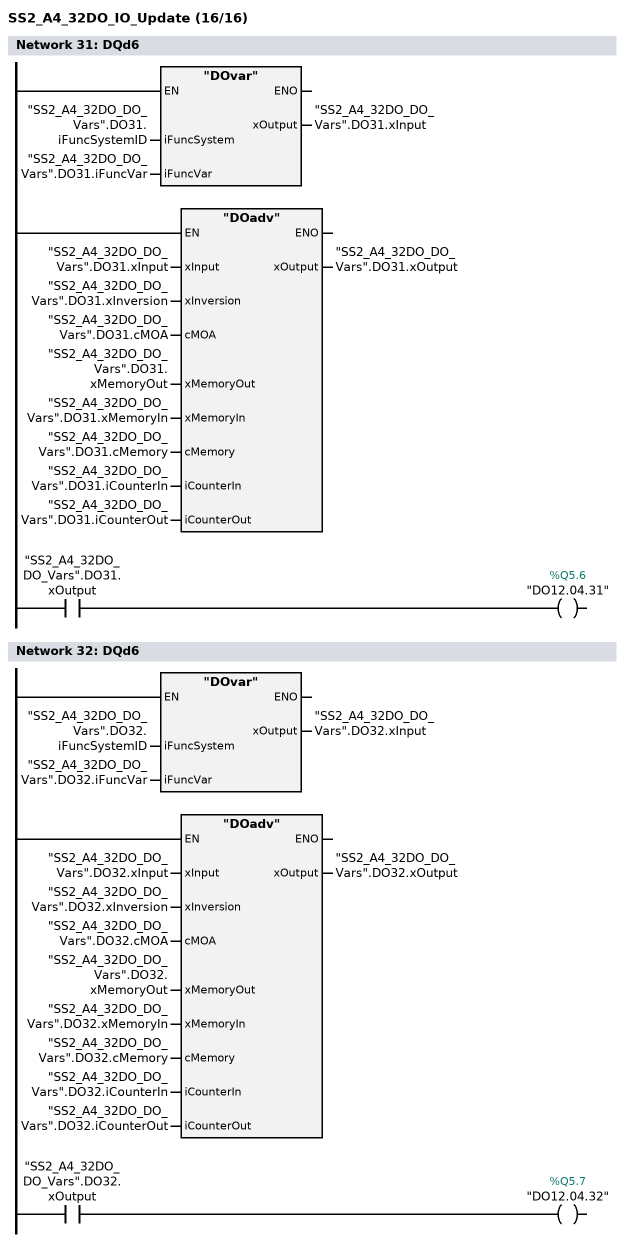
   RUNG wire#powerrail
      "DOvar"(iFuncSystem := "SS2_A4_32DO_DO_Vars".DO31.iFuncSystemID, iFuncVar := "SS2_A4_32DO_DO_Vars".DO31.iFuncVar, xOutput => "SS2_A4_32DO_DO_Vars".DO31.xInput)
   END_RUNG
   RUNG wire#powerrail
      "DOadv"(xInput := "SS2_A4_32DO_DO_Vars".DO31.xInput, xInversion := "SS2_A4_32DO_DO_Vars".DO31.xInversion, cMOA := "SS2_A4_32DO_DO_Vars".DO31.cMOA, xMemoryOut := "SS2_A4_32DO_DO_Vars".DO31.xMemoryOut, xMemoryIn := "SS2_A4_32DO_DO_Vars".DO31.xMemoryIn, cMemory := "SS2_A4_32DO_DO_Vars".DO31.cMemory, iCounterIn := "SS2_A4_32DO_DO_Vars".DO31.iCounterIn, iCounterOut := "SS2_A4_32DO_DO_Vars".DO31.iCounterOut, xOutput => "SS2_A4_32DO_DO_Vars".DO31.xOutput)
   END_RUNG
   RUNG wire#powerrail
      Contact( "SS2_A4_32DO_DO_Vars".DO31.xOutput )
      Coil( "DO12.04.31" )
   END_RUNG
   // the same network as SCL:
   "DOvar"(iFuncSystem := "SS2_A4_32DO_DO_Vars".DO31.iFuncSystemID,
           iFuncVar := "SS2_A4_32DO_DO_Vars".DO31.iFuncVar,
           xOutput => "SS2_A4_32DO_DO_Vars".DO31.xInput);
   "DOadv"(xInput := "SS2_A4_32DO_DO_Vars".DO31.xInput,
           xInversion := "SS2_A4_32DO_DO_Vars".DO31.xInversion,
           cMOA := "SS2_A4_32DO_DO_Vars".DO31.cMOA,
           xMemoryOut := "SS2_A4_32DO_DO_Vars".DO31.xMemoryOut,
           xMemoryIn := "SS2_A4_32DO_DO_Vars".DO31.xMemoryIn,
           cMemory := "SS2_A4_32DO_DO_Vars".DO31.cMemory,
           iCounterIn := "SS2_A4_32DO_DO_Vars".DO31.iCounterIn,
           iCounterOut := "SS2_A4_32DO_DO_Vars".DO31.iCounterOut,
           xOutput => "SS2_A4_32DO_DO_Vars".DO31.xOutput);
   "DO12.04.31" := "SS2_A4_32DO_DO_Vars".DO31.xOutput;
END_REGION

REGION Network 32: DQd6
   RUNG wire#powerrail
      "DOvar"(iFuncSystem := "SS2_A4_32DO_DO_Vars".DO32.iFuncSystemID, iFuncVar := "SS2_A4_32DO_DO_Vars".DO32.iFuncVar, xOutput => "SS2_A4_32DO_DO_Vars".DO32.xInput)
   END_RUNG
   RUNG wire#powerrail
      "DOadv"(xInput := "SS2_A4_32DO_DO_Vars".DO32.xInput, xInversion := "SS2_A4_32DO_DO_Vars".DO32.xInversion, cMOA := "SS2_A4_32DO_DO_Vars".DO32.cMOA, xMemoryOut := "SS2_A4_32DO_DO_Vars".DO32.xMemoryOut, xMemoryIn := "SS2_A4_32DO_DO_Vars".DO32.xMemoryIn, cMemory := "SS2_A4_32DO_DO_Vars".DO32.cMemory, iCounterIn := "SS2_A4_32DO_DO_Vars".DO32.iCounterIn, iCounterOut := "SS2_A4_32DO_DO_Vars".DO32.iCounterOut, xOutput => "SS2_A4_32DO_DO_Vars".DO32.xOutput)
   END_RUNG
   RUNG wire#powerrail
      Contact( "SS2_A4_32DO_DO_Vars".DO32.xOutput )
      Coil( "DO12.04.32" )
   END_RUNG
   // the same network as SCL:
   "DOvar"(iFuncSystem := "SS2_A4_32DO_DO_Vars".DO32.iFuncSystemID,
           iFuncVar := "SS2_A4_32DO_DO_Vars".DO32.iFuncVar,
           xOutput => "SS2_A4_32DO_DO_Vars".DO32.xInput);
   "DOadv"(xInput := "SS2_A4_32DO_DO_Vars".DO32.xInput,
           xInversion := "SS2_A4_32DO_DO_Vars".DO32.xInversion,
           cMOA := "SS2_A4_32DO_DO_Vars".DO32.cMOA,
           xMemoryOut := "SS2_A4_32DO_DO_Vars".DO32.xMemoryOut,
           xMemoryIn := "SS2_A4_32DO_DO_Vars".DO32.xMemoryIn,
           cMemory := "SS2_A4_32DO_DO_Vars".DO32.cMemory,
           iCounterIn := "SS2_A4_32DO_DO_Vars".DO32.iCounterIn,
           iCounterOut := "SS2_A4_32DO_DO_Vars".DO32.iCounterOut,
           xOutput => "SS2_A4_32DO_DO_Vars".DO32.xOutput);
   "DO12.04.32" := "SS2_A4_32DO_DO_Vars".DO32.xOutput;
END_REGION
END_FUNCTION

FUNCTION "SS2_A5_16DI_IO_Update" : Void   // FC11160, LAD
{ S7_Optimized_Access := 'TRUE' }
VERSION : 0.1
// stored: AutoNumber false, IsIECCheckEnabled false, SetENOAutomatically false, UDAEnableTagReadback false
BEGIN

REGION Network 1: DIa0
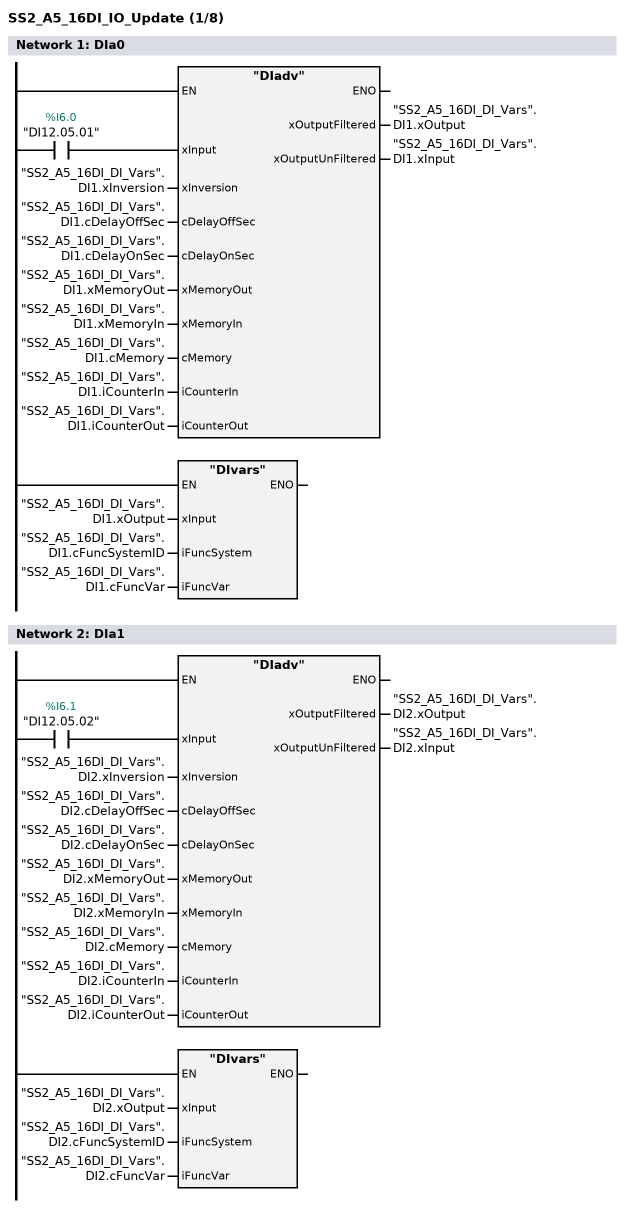
   RUNG wire#powerrail
      "DIadv"(xInput := wire#w1, xInversion := "SS2_A5_16DI_DI_Vars".DI1.xInversion, cDelayOffSec := "SS2_A5_16DI_DI_Vars".DI1.cDelayOffSec, cDelayOnSec := "SS2_A5_16DI_DI_Vars".DI1.cDelayOnSec, xMemoryOut := "SS2_A5_16DI_DI_Vars".DI1.xMemoryOut, xMemoryIn := "SS2_A5_16DI_DI_Vars".DI1.xMemoryIn, cMemory := "SS2_A5_16DI_DI_Vars".DI1.cMemory, xOutputFiltered => "SS2_A5_16DI_DI_Vars".DI1.xOutput, xOutputUnFiltered => "SS2_A5_16DI_DI_Vars".DI1.xInput, iCounterIn := "SS2_A5_16DI_DI_Vars".DI1.iCounterIn, iCounterOut := "SS2_A5_16DI_DI_Vars".DI1.iCounterOut)
   END_RUNG
   RUNG wire#powerrail
      Contact( "DI12.05.01" )
   END_RUNG wire#w1
   RUNG wire#powerrail
      "DIvars"(xInput := "SS2_A5_16DI_DI_Vars".DI1.xOutput, iFuncSystem := "SS2_A5_16DI_DI_Vars".DI1.cFuncSystemID, iFuncVar := "SS2_A5_16DI_DI_Vars".DI1.cFuncVar)
   END_RUNG
   // the same network as SCL:
   "DIadv"(xInput := "DI12.05.01",
           xInversion := "SS2_A5_16DI_DI_Vars".DI1.xInversion,
           cDelayOffSec := "SS2_A5_16DI_DI_Vars".DI1.cDelayOffSec,
           cDelayOnSec := "SS2_A5_16DI_DI_Vars".DI1.cDelayOnSec,
           xMemoryOut := "SS2_A5_16DI_DI_Vars".DI1.xMemoryOut,
           xMemoryIn := "SS2_A5_16DI_DI_Vars".DI1.xMemoryIn,
           cMemory := "SS2_A5_16DI_DI_Vars".DI1.cMemory,
           iCounterIn := "SS2_A5_16DI_DI_Vars".DI1.iCounterIn,
           iCounterOut := "SS2_A5_16DI_DI_Vars".DI1.iCounterOut,
           xOutputFiltered => "SS2_A5_16DI_DI_Vars".DI1.xOutput,
           xOutputUnFiltered => "SS2_A5_16DI_DI_Vars".DI1.xInput);
   "DIvars"(xInput := "SS2_A5_16DI_DI_Vars".DI1.xOutput,
            iFuncSystem := "SS2_A5_16DI_DI_Vars".DI1.cFuncSystemID,
            iFuncVar := "SS2_A5_16DI_DI_Vars".DI1.cFuncVar);
END_REGION

REGION Network 2: DIa1
   RUNG wire#powerrail
      "DIadv"(xInput := wire#w1, xInversion := "SS2_A5_16DI_DI_Vars".DI2.xInversion, cDelayOffSec := "SS2_A5_16DI_DI_Vars".DI2.cDelayOffSec, cDelayOnSec := "SS2_A5_16DI_DI_Vars".DI2.cDelayOnSec, xMemoryOut := "SS2_A5_16DI_DI_Vars".DI2.xMemoryOut, xMemoryIn := "SS2_A5_16DI_DI_Vars".DI2.xMemoryIn, cMemory := "SS2_A5_16DI_DI_Vars".DI2.cMemory, xOutputFiltered => "SS2_A5_16DI_DI_Vars".DI2.xOutput, xOutputUnFiltered => "SS2_A5_16DI_DI_Vars".DI2.xInput, iCounterIn := "SS2_A5_16DI_DI_Vars".DI2.iCounterIn, iCounterOut := "SS2_A5_16DI_DI_Vars".DI2.iCounterOut)
   END_RUNG
   RUNG wire#powerrail
      Contact( "DI12.05.02" )
   END_RUNG wire#w1
   RUNG wire#powerrail
      "DIvars"(xInput := "SS2_A5_16DI_DI_Vars".DI2.xOutput, iFuncSystem := "SS2_A5_16DI_DI_Vars".DI2.cFuncSystemID, iFuncVar := "SS2_A5_16DI_DI_Vars".DI2.cFuncVar)
   END_RUNG
   // the same network as SCL:
   "DIadv"(xInput := "DI12.05.02",
           xInversion := "SS2_A5_16DI_DI_Vars".DI2.xInversion,
           cDelayOffSec := "SS2_A5_16DI_DI_Vars".DI2.cDelayOffSec,
           cDelayOnSec := "SS2_A5_16DI_DI_Vars".DI2.cDelayOnSec,
           xMemoryOut := "SS2_A5_16DI_DI_Vars".DI2.xMemoryOut,
           xMemoryIn := "SS2_A5_16DI_DI_Vars".DI2.xMemoryIn,
           cMemory := "SS2_A5_16DI_DI_Vars".DI2.cMemory,
           iCounterIn := "SS2_A5_16DI_DI_Vars".DI2.iCounterIn,
           iCounterOut := "SS2_A5_16DI_DI_Vars".DI2.iCounterOut,
           xOutputFiltered => "SS2_A5_16DI_DI_Vars".DI2.xOutput,
           xOutputUnFiltered => "SS2_A5_16DI_DI_Vars".DI2.xInput);
   "DIvars"(xInput := "SS2_A5_16DI_DI_Vars".DI2.xOutput,
            iFuncSystem := "SS2_A5_16DI_DI_Vars".DI2.cFuncSystemID,
            iFuncVar := "SS2_A5_16DI_DI_Vars".DI2.cFuncVar);
END_REGION

REGION Network 3: DIa2
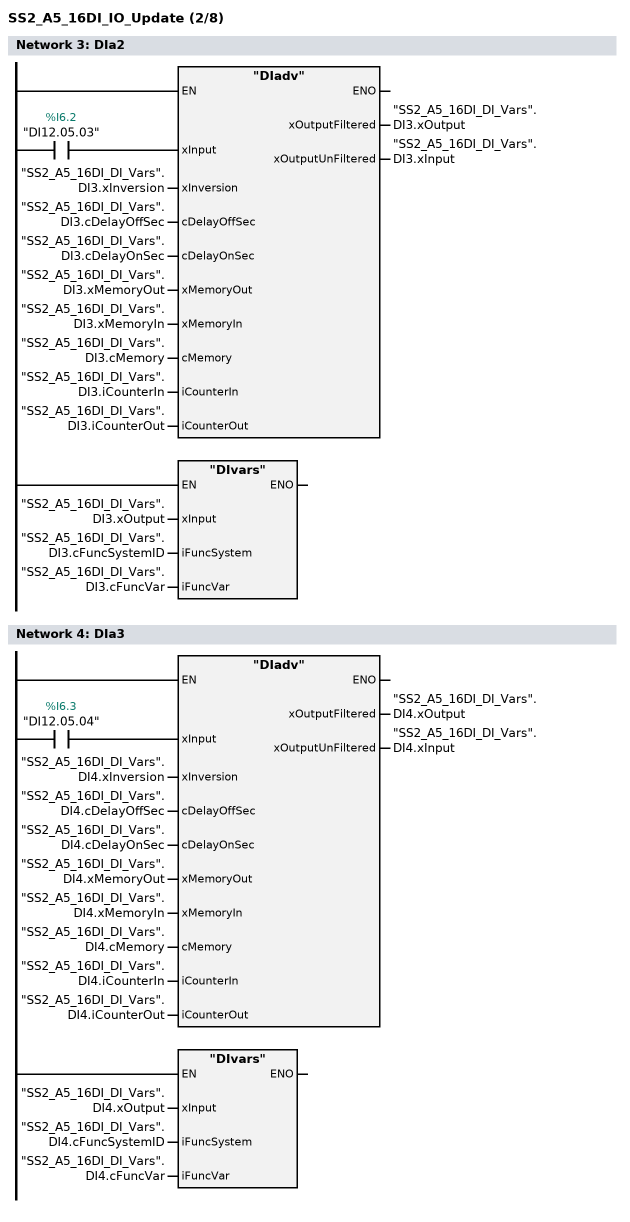
   RUNG wire#powerrail
      "DIadv"(xInput := wire#w1, xInversion := "SS2_A5_16DI_DI_Vars".DI3.xInversion, cDelayOffSec := "SS2_A5_16DI_DI_Vars".DI3.cDelayOffSec, cDelayOnSec := "SS2_A5_16DI_DI_Vars".DI3.cDelayOnSec, xMemoryOut := "SS2_A5_16DI_DI_Vars".DI3.xMemoryOut, xMemoryIn := "SS2_A5_16DI_DI_Vars".DI3.xMemoryIn, cMemory := "SS2_A5_16DI_DI_Vars".DI3.cMemory, xOutputFiltered => "SS2_A5_16DI_DI_Vars".DI3.xOutput, xOutputUnFiltered => "SS2_A5_16DI_DI_Vars".DI3.xInput, iCounterIn := "SS2_A5_16DI_DI_Vars".DI3.iCounterIn, iCounterOut := "SS2_A5_16DI_DI_Vars".DI3.iCounterOut)
   END_RUNG
   RUNG wire#powerrail
      Contact( "DI12.05.03" )
   END_RUNG wire#w1
   RUNG wire#powerrail
      "DIvars"(xInput := "SS2_A5_16DI_DI_Vars".DI3.xOutput, iFuncSystem := "SS2_A5_16DI_DI_Vars".DI3.cFuncSystemID, iFuncVar := "SS2_A5_16DI_DI_Vars".DI3.cFuncVar)
   END_RUNG
   // the same network as SCL:
   "DIadv"(xInput := "DI12.05.03",
           xInversion := "SS2_A5_16DI_DI_Vars".DI3.xInversion,
           cDelayOffSec := "SS2_A5_16DI_DI_Vars".DI3.cDelayOffSec,
           cDelayOnSec := "SS2_A5_16DI_DI_Vars".DI3.cDelayOnSec,
           xMemoryOut := "SS2_A5_16DI_DI_Vars".DI3.xMemoryOut,
           xMemoryIn := "SS2_A5_16DI_DI_Vars".DI3.xMemoryIn,
           cMemory := "SS2_A5_16DI_DI_Vars".DI3.cMemory,
           iCounterIn := "SS2_A5_16DI_DI_Vars".DI3.iCounterIn,
           iCounterOut := "SS2_A5_16DI_DI_Vars".DI3.iCounterOut,
           xOutputFiltered => "SS2_A5_16DI_DI_Vars".DI3.xOutput,
           xOutputUnFiltered => "SS2_A5_16DI_DI_Vars".DI3.xInput);
   "DIvars"(xInput := "SS2_A5_16DI_DI_Vars".DI3.xOutput,
            iFuncSystem := "SS2_A5_16DI_DI_Vars".DI3.cFuncSystemID,
            iFuncVar := "SS2_A5_16DI_DI_Vars".DI3.cFuncVar);
END_REGION

REGION Network 4: DIa3
   RUNG wire#powerrail
      "DIadv"(xInput := wire#w1, xInversion := "SS2_A5_16DI_DI_Vars".DI4.xInversion, cDelayOffSec := "SS2_A5_16DI_DI_Vars".DI4.cDelayOffSec, cDelayOnSec := "SS2_A5_16DI_DI_Vars".DI4.cDelayOnSec, xMemoryOut := "SS2_A5_16DI_DI_Vars".DI4.xMemoryOut, xMemoryIn := "SS2_A5_16DI_DI_Vars".DI4.xMemoryIn, cMemory := "SS2_A5_16DI_DI_Vars".DI4.cMemory, xOutputFiltered => "SS2_A5_16DI_DI_Vars".DI4.xOutput, xOutputUnFiltered => "SS2_A5_16DI_DI_Vars".DI4.xInput, iCounterIn := "SS2_A5_16DI_DI_Vars".DI4.iCounterIn, iCounterOut := "SS2_A5_16DI_DI_Vars".DI4.iCounterOut)
   END_RUNG
   RUNG wire#powerrail
      Contact( "DI12.05.04" )
   END_RUNG wire#w1
   RUNG wire#powerrail
      "DIvars"(xInput := "SS2_A5_16DI_DI_Vars".DI4.xOutput, iFuncSystem := "SS2_A5_16DI_DI_Vars".DI4.cFuncSystemID, iFuncVar := "SS2_A5_16DI_DI_Vars".DI4.cFuncVar)
   END_RUNG
   // the same network as SCL:
   "DIadv"(xInput := "DI12.05.04",
           xInversion := "SS2_A5_16DI_DI_Vars".DI4.xInversion,
           cDelayOffSec := "SS2_A5_16DI_DI_Vars".DI4.cDelayOffSec,
           cDelayOnSec := "SS2_A5_16DI_DI_Vars".DI4.cDelayOnSec,
           xMemoryOut := "SS2_A5_16DI_DI_Vars".DI4.xMemoryOut,
           xMemoryIn := "SS2_A5_16DI_DI_Vars".DI4.xMemoryIn,
           cMemory := "SS2_A5_16DI_DI_Vars".DI4.cMemory,
           iCounterIn := "SS2_A5_16DI_DI_Vars".DI4.iCounterIn,
           iCounterOut := "SS2_A5_16DI_DI_Vars".DI4.iCounterOut,
           xOutputFiltered => "SS2_A5_16DI_DI_Vars".DI4.xOutput,
           xOutputUnFiltered => "SS2_A5_16DI_DI_Vars".DI4.xInput);
   "DIvars"(xInput := "SS2_A5_16DI_DI_Vars".DI4.xOutput,
            iFuncSystem := "SS2_A5_16DI_DI_Vars".DI4.cFuncSystemID,
            iFuncVar := "SS2_A5_16DI_DI_Vars".DI4.cFuncVar);
END_REGION

REGION Network 5: DIa4
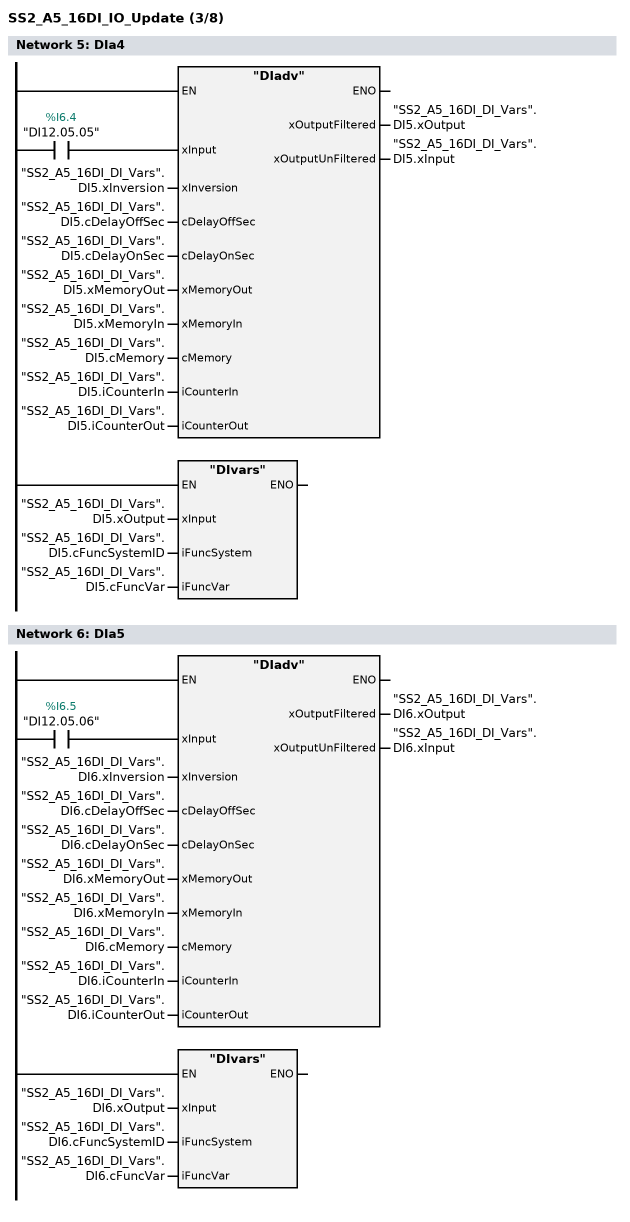
   RUNG wire#powerrail
      "DIadv"(xInput := wire#w1, xInversion := "SS2_A5_16DI_DI_Vars".DI5.xInversion, cDelayOffSec := "SS2_A5_16DI_DI_Vars".DI5.cDelayOffSec, cDelayOnSec := "SS2_A5_16DI_DI_Vars".DI5.cDelayOnSec, xMemoryOut := "SS2_A5_16DI_DI_Vars".DI5.xMemoryOut, xMemoryIn := "SS2_A5_16DI_DI_Vars".DI5.xMemoryIn, cMemory := "SS2_A5_16DI_DI_Vars".DI5.cMemory, xOutputFiltered => "SS2_A5_16DI_DI_Vars".DI5.xOutput, xOutputUnFiltered => "SS2_A5_16DI_DI_Vars".DI5.xInput, iCounterIn := "SS2_A5_16DI_DI_Vars".DI5.iCounterIn, iCounterOut := "SS2_A5_16DI_DI_Vars".DI5.iCounterOut)
   END_RUNG
   RUNG wire#powerrail
      Contact( "DI12.05.05" )
   END_RUNG wire#w1
   RUNG wire#powerrail
      "DIvars"(xInput := "SS2_A5_16DI_DI_Vars".DI5.xOutput, iFuncSystem := "SS2_A5_16DI_DI_Vars".DI5.cFuncSystemID, iFuncVar := "SS2_A5_16DI_DI_Vars".DI5.cFuncVar)
   END_RUNG
   // the same network as SCL:
   "DIadv"(xInput := "DI12.05.05",
           xInversion := "SS2_A5_16DI_DI_Vars".DI5.xInversion,
           cDelayOffSec := "SS2_A5_16DI_DI_Vars".DI5.cDelayOffSec,
           cDelayOnSec := "SS2_A5_16DI_DI_Vars".DI5.cDelayOnSec,
           xMemoryOut := "SS2_A5_16DI_DI_Vars".DI5.xMemoryOut,
           xMemoryIn := "SS2_A5_16DI_DI_Vars".DI5.xMemoryIn,
           cMemory := "SS2_A5_16DI_DI_Vars".DI5.cMemory,
           iCounterIn := "SS2_A5_16DI_DI_Vars".DI5.iCounterIn,
           iCounterOut := "SS2_A5_16DI_DI_Vars".DI5.iCounterOut,
           xOutputFiltered => "SS2_A5_16DI_DI_Vars".DI5.xOutput,
           xOutputUnFiltered => "SS2_A5_16DI_DI_Vars".DI5.xInput);
   "DIvars"(xInput := "SS2_A5_16DI_DI_Vars".DI5.xOutput,
            iFuncSystem := "SS2_A5_16DI_DI_Vars".DI5.cFuncSystemID,
            iFuncVar := "SS2_A5_16DI_DI_Vars".DI5.cFuncVar);
END_REGION

REGION Network 6: DIa5
   RUNG wire#powerrail
      "DIadv"(xInput := wire#w1, xInversion := "SS2_A5_16DI_DI_Vars".DI6.xInversion, cDelayOffSec := "SS2_A5_16DI_DI_Vars".DI6.cDelayOffSec, cDelayOnSec := "SS2_A5_16DI_DI_Vars".DI6.cDelayOnSec, xMemoryOut := "SS2_A5_16DI_DI_Vars".DI6.xMemoryOut, xMemoryIn := "SS2_A5_16DI_DI_Vars".DI6.xMemoryIn, cMemory := "SS2_A5_16DI_DI_Vars".DI6.cMemory, xOutputFiltered => "SS2_A5_16DI_DI_Vars".DI6.xOutput, xOutputUnFiltered => "SS2_A5_16DI_DI_Vars".DI6.xInput, iCounterIn := "SS2_A5_16DI_DI_Vars".DI6.iCounterIn, iCounterOut := "SS2_A5_16DI_DI_Vars".DI6.iCounterOut)
   END_RUNG
   RUNG wire#powerrail
      Contact( "DI12.05.06" )
   END_RUNG wire#w1
   RUNG wire#powerrail
      "DIvars"(xInput := "SS2_A5_16DI_DI_Vars".DI6.xOutput, iFuncSystem := "SS2_A5_16DI_DI_Vars".DI6.cFuncSystemID, iFuncVar := "SS2_A5_16DI_DI_Vars".DI6.cFuncVar)
   END_RUNG
   // the same network as SCL:
   "DIadv"(xInput := "DI12.05.06",
           xInversion := "SS2_A5_16DI_DI_Vars".DI6.xInversion,
           cDelayOffSec := "SS2_A5_16DI_DI_Vars".DI6.cDelayOffSec,
           cDelayOnSec := "SS2_A5_16DI_DI_Vars".DI6.cDelayOnSec,
           xMemoryOut := "SS2_A5_16DI_DI_Vars".DI6.xMemoryOut,
           xMemoryIn := "SS2_A5_16DI_DI_Vars".DI6.xMemoryIn,
           cMemory := "SS2_A5_16DI_DI_Vars".DI6.cMemory,
           iCounterIn := "SS2_A5_16DI_DI_Vars".DI6.iCounterIn,
           iCounterOut := "SS2_A5_16DI_DI_Vars".DI6.iCounterOut,
           xOutputFiltered => "SS2_A5_16DI_DI_Vars".DI6.xOutput,
           xOutputUnFiltered => "SS2_A5_16DI_DI_Vars".DI6.xInput);
   "DIvars"(xInput := "SS2_A5_16DI_DI_Vars".DI6.xOutput,
            iFuncSystem := "SS2_A5_16DI_DI_Vars".DI6.cFuncSystemID,
            iFuncVar := "SS2_A5_16DI_DI_Vars".DI6.cFuncVar);
END_REGION

REGION Network 7: DIa6
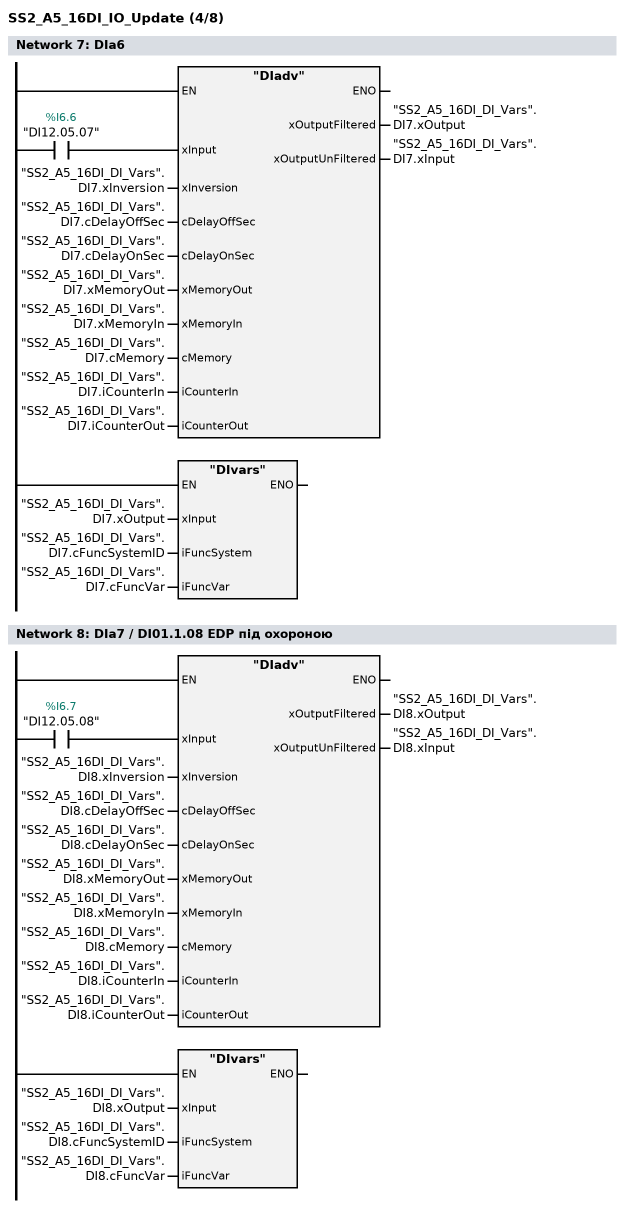
   RUNG wire#powerrail
      "DIadv"(xInput := wire#w1, xInversion := "SS2_A5_16DI_DI_Vars".DI7.xInversion, cDelayOffSec := "SS2_A5_16DI_DI_Vars".DI7.cDelayOffSec, cDelayOnSec := "SS2_A5_16DI_DI_Vars".DI7.cDelayOnSec, xMemoryOut := "SS2_A5_16DI_DI_Vars".DI7.xMemoryOut, xMemoryIn := "SS2_A5_16DI_DI_Vars".DI7.xMemoryIn, cMemory := "SS2_A5_16DI_DI_Vars".DI7.cMemory, xOutputFiltered => "SS2_A5_16DI_DI_Vars".DI7.xOutput, xOutputUnFiltered => "SS2_A5_16DI_DI_Vars".DI7.xInput, iCounterIn := "SS2_A5_16DI_DI_Vars".DI7.iCounterIn, iCounterOut := "SS2_A5_16DI_DI_Vars".DI7.iCounterOut)
   END_RUNG
   RUNG wire#powerrail
      Contact( "DI12.05.07" )
   END_RUNG wire#w1
   RUNG wire#powerrail
      "DIvars"(xInput := "SS2_A5_16DI_DI_Vars".DI7.xOutput, iFuncSystem := "SS2_A5_16DI_DI_Vars".DI7.cFuncSystemID, iFuncVar := "SS2_A5_16DI_DI_Vars".DI7.cFuncVar)
   END_RUNG
   // the same network as SCL:
   "DIadv"(xInput := "DI12.05.07",
           xInversion := "SS2_A5_16DI_DI_Vars".DI7.xInversion,
           cDelayOffSec := "SS2_A5_16DI_DI_Vars".DI7.cDelayOffSec,
           cDelayOnSec := "SS2_A5_16DI_DI_Vars".DI7.cDelayOnSec,
           xMemoryOut := "SS2_A5_16DI_DI_Vars".DI7.xMemoryOut,
           xMemoryIn := "SS2_A5_16DI_DI_Vars".DI7.xMemoryIn,
           cMemory := "SS2_A5_16DI_DI_Vars".DI7.cMemory,
           iCounterIn := "SS2_A5_16DI_DI_Vars".DI7.iCounterIn,
           iCounterOut := "SS2_A5_16DI_DI_Vars".DI7.iCounterOut,
           xOutputFiltered => "SS2_A5_16DI_DI_Vars".DI7.xOutput,
           xOutputUnFiltered => "SS2_A5_16DI_DI_Vars".DI7.xInput);
   "DIvars"(xInput := "SS2_A5_16DI_DI_Vars".DI7.xOutput,
            iFuncSystem := "SS2_A5_16DI_DI_Vars".DI7.cFuncSystemID,
            iFuncVar := "SS2_A5_16DI_DI_Vars".DI7.cFuncVar);
END_REGION

REGION Network 8: DIa7 / DI01.1.08 EDP під охороною
   RUNG wire#powerrail
      "DIadv"(xInput := wire#w1, xInversion := "SS2_A5_16DI_DI_Vars".DI8.xInversion, cDelayOffSec := "SS2_A5_16DI_DI_Vars".DI8.cDelayOffSec, cDelayOnSec := "SS2_A5_16DI_DI_Vars".DI8.cDelayOnSec, xMemoryOut := "SS2_A5_16DI_DI_Vars".DI8.xMemoryOut, xMemoryIn := "SS2_A5_16DI_DI_Vars".DI8.xMemoryIn, cMemory := "SS2_A5_16DI_DI_Vars".DI8.cMemory, xOutputFiltered => "SS2_A5_16DI_DI_Vars".DI8.xOutput, xOutputUnFiltered => "SS2_A5_16DI_DI_Vars".DI8.xInput, iCounterIn := "SS2_A5_16DI_DI_Vars".DI8.iCounterIn, iCounterOut := "SS2_A5_16DI_DI_Vars".DI8.iCounterOut)
   END_RUNG
   RUNG wire#powerrail
      Contact( "DI12.05.08" )
   END_RUNG wire#w1
   RUNG wire#powerrail
      "DIvars"(xInput := "SS2_A5_16DI_DI_Vars".DI8.xOutput, iFuncSystem := "SS2_A5_16DI_DI_Vars".DI8.cFuncSystemID, iFuncVar := "SS2_A5_16DI_DI_Vars".DI8.cFuncVar)
   END_RUNG
   // the same network as SCL:
   "DIadv"(xInput := "DI12.05.08",
           xInversion := "SS2_A5_16DI_DI_Vars".DI8.xInversion,
           cDelayOffSec := "SS2_A5_16DI_DI_Vars".DI8.cDelayOffSec,
           cDelayOnSec := "SS2_A5_16DI_DI_Vars".DI8.cDelayOnSec,
           xMemoryOut := "SS2_A5_16DI_DI_Vars".DI8.xMemoryOut,
           xMemoryIn := "SS2_A5_16DI_DI_Vars".DI8.xMemoryIn,
           cMemory := "SS2_A5_16DI_DI_Vars".DI8.cMemory,
           iCounterIn := "SS2_A5_16DI_DI_Vars".DI8.iCounterIn,
           iCounterOut := "SS2_A5_16DI_DI_Vars".DI8.iCounterOut,
           xOutputFiltered => "SS2_A5_16DI_DI_Vars".DI8.xOutput,
           xOutputUnFiltered => "SS2_A5_16DI_DI_Vars".DI8.xInput);
   "DIvars"(xInput := "SS2_A5_16DI_DI_Vars".DI8.xOutput,
            iFuncSystem := "SS2_A5_16DI_DI_Vars".DI8.cFuncSystemID,
            iFuncVar := "SS2_A5_16DI_DI_Vars".DI8.cFuncVar);
END_REGION

REGION Network 9: DIb0 / DI01.1.08 EDP під охороною
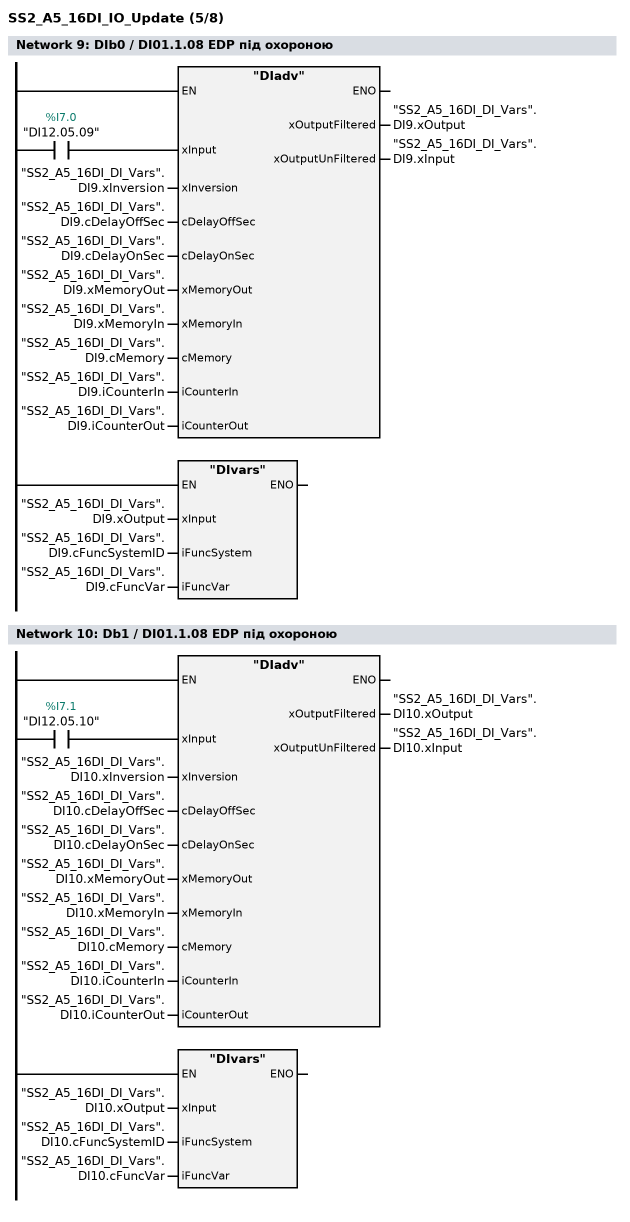
   RUNG wire#powerrail
      "DIadv"(xInput := wire#w1, xInversion := "SS2_A5_16DI_DI_Vars".DI9.xInversion, cDelayOffSec := "SS2_A5_16DI_DI_Vars".DI9.cDelayOffSec, cDelayOnSec := "SS2_A5_16DI_DI_Vars".DI9.cDelayOnSec, xMemoryOut := "SS2_A5_16DI_DI_Vars".DI9.xMemoryOut, xMemoryIn := "SS2_A5_16DI_DI_Vars".DI9.xMemoryIn, cMemory := "SS2_A5_16DI_DI_Vars".DI9.cMemory, xOutputFiltered => "SS2_A5_16DI_DI_Vars".DI9.xOutput, xOutputUnFiltered => "SS2_A5_16DI_DI_Vars".DI9.xInput, iCounterIn := "SS2_A5_16DI_DI_Vars".DI9.iCounterIn, iCounterOut := "SS2_A5_16DI_DI_Vars".DI9.iCounterOut)
   END_RUNG
   RUNG wire#powerrail
      Contact( "DI12.05.09" )
   END_RUNG wire#w1
   RUNG wire#powerrail
      "DIvars"(xInput := "SS2_A5_16DI_DI_Vars".DI9.xOutput, iFuncSystem := "SS2_A5_16DI_DI_Vars".DI9.cFuncSystemID, iFuncVar := "SS2_A5_16DI_DI_Vars".DI9.cFuncVar)
   END_RUNG
   // the same network as SCL:
   "DIadv"(xInput := "DI12.05.09",
           xInversion := "SS2_A5_16DI_DI_Vars".DI9.xInversion,
           cDelayOffSec := "SS2_A5_16DI_DI_Vars".DI9.cDelayOffSec,
           cDelayOnSec := "SS2_A5_16DI_DI_Vars".DI9.cDelayOnSec,
           xMemoryOut := "SS2_A5_16DI_DI_Vars".DI9.xMemoryOut,
           xMemoryIn := "SS2_A5_16DI_DI_Vars".DI9.xMemoryIn,
           cMemory := "SS2_A5_16DI_DI_Vars".DI9.cMemory,
           iCounterIn := "SS2_A5_16DI_DI_Vars".DI9.iCounterIn,
           iCounterOut := "SS2_A5_16DI_DI_Vars".DI9.iCounterOut,
           xOutputFiltered => "SS2_A5_16DI_DI_Vars".DI9.xOutput,
           xOutputUnFiltered => "SS2_A5_16DI_DI_Vars".DI9.xInput);
   "DIvars"(xInput := "SS2_A5_16DI_DI_Vars".DI9.xOutput,
            iFuncSystem := "SS2_A5_16DI_DI_Vars".DI9.cFuncSystemID,
            iFuncVar := "SS2_A5_16DI_DI_Vars".DI9.cFuncVar);
END_REGION

REGION Network 10: Db1 / DI01.1.08 EDP під охороною
   RUNG wire#powerrail
      "DIadv"(xInput := wire#w1, xInversion := "SS2_A5_16DI_DI_Vars".DI10.xInversion, cDelayOffSec := "SS2_A5_16DI_DI_Vars".DI10.cDelayOffSec, cDelayOnSec := "SS2_A5_16DI_DI_Vars".DI10.cDelayOnSec, xMemoryOut := "SS2_A5_16DI_DI_Vars".DI10.xMemoryOut, xMemoryIn := "SS2_A5_16DI_DI_Vars".DI10.xMemoryIn, cMemory := "SS2_A5_16DI_DI_Vars".DI10.cMemory, xOutputFiltered => "SS2_A5_16DI_DI_Vars".DI10.xOutput, xOutputUnFiltered => "SS2_A5_16DI_DI_Vars".DI10.xInput, iCounterIn := "SS2_A5_16DI_DI_Vars".DI10.iCounterIn, iCounterOut := "SS2_A5_16DI_DI_Vars".DI10.iCounterOut)
   END_RUNG
   RUNG wire#powerrail
      Contact( "DI12.05.10" )
   END_RUNG wire#w1
   RUNG wire#powerrail
      "DIvars"(xInput := "SS2_A5_16DI_DI_Vars".DI10.xOutput, iFuncSystem := "SS2_A5_16DI_DI_Vars".DI10.cFuncSystemID, iFuncVar := "SS2_A5_16DI_DI_Vars".DI10.cFuncVar)
   END_RUNG
   // the same network as SCL:
   "DIadv"(xInput := "DI12.05.10",
           xInversion := "SS2_A5_16DI_DI_Vars".DI10.xInversion,
           cDelayOffSec := "SS2_A5_16DI_DI_Vars".DI10.cDelayOffSec,
           cDelayOnSec := "SS2_A5_16DI_DI_Vars".DI10.cDelayOnSec,
           xMemoryOut := "SS2_A5_16DI_DI_Vars".DI10.xMemoryOut,
           xMemoryIn := "SS2_A5_16DI_DI_Vars".DI10.xMemoryIn,
           cMemory := "SS2_A5_16DI_DI_Vars".DI10.cMemory,
           iCounterIn := "SS2_A5_16DI_DI_Vars".DI10.iCounterIn,
           iCounterOut := "SS2_A5_16DI_DI_Vars".DI10.iCounterOut,
           xOutputFiltered => "SS2_A5_16DI_DI_Vars".DI10.xOutput,
           xOutputUnFiltered => "SS2_A5_16DI_DI_Vars".DI10.xInput);
   "DIvars"(xInput := "SS2_A5_16DI_DI_Vars".DI10.xOutput,
            iFuncSystem := "SS2_A5_16DI_DI_Vars".DI10.cFuncSystemID,
            iFuncVar := "SS2_A5_16DI_DI_Vars".DI10.cFuncVar);
END_REGION

REGION Network 11: DIb2 / DI01.1.08 EDP під охороною
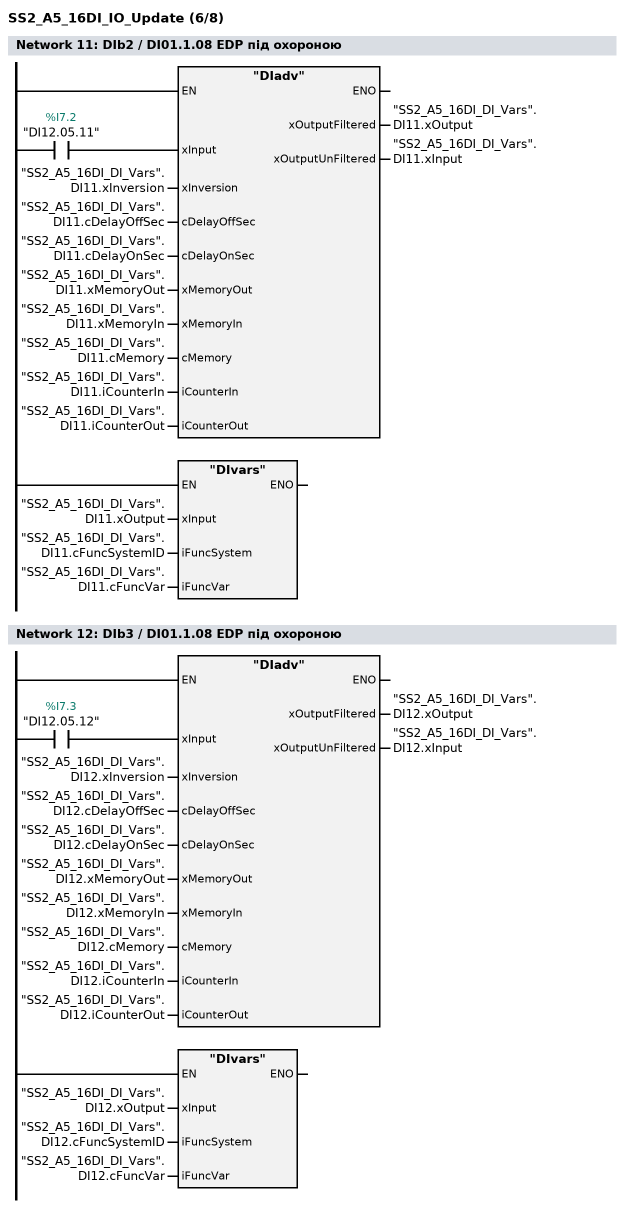
   RUNG wire#powerrail
      "DIadv"(xInput := wire#w1, xInversion := "SS2_A5_16DI_DI_Vars".DI11.xInversion, cDelayOffSec := "SS2_A5_16DI_DI_Vars".DI11.cDelayOffSec, cDelayOnSec := "SS2_A5_16DI_DI_Vars".DI11.cDelayOnSec, xMemoryOut := "SS2_A5_16DI_DI_Vars".DI11.xMemoryOut, xMemoryIn := "SS2_A5_16DI_DI_Vars".DI11.xMemoryIn, cMemory := "SS2_A5_16DI_DI_Vars".DI11.cMemory, xOutputFiltered => "SS2_A5_16DI_DI_Vars".DI11.xOutput, xOutputUnFiltered => "SS2_A5_16DI_DI_Vars".DI11.xInput, iCounterIn := "SS2_A5_16DI_DI_Vars".DI11.iCounterIn, iCounterOut := "SS2_A5_16DI_DI_Vars".DI11.iCounterOut)
   END_RUNG
   RUNG wire#powerrail
      Contact( "DI12.05.11" )
   END_RUNG wire#w1
   RUNG wire#powerrail
      "DIvars"(xInput := "SS2_A5_16DI_DI_Vars".DI11.xOutput, iFuncSystem := "SS2_A5_16DI_DI_Vars".DI11.cFuncSystemID, iFuncVar := "SS2_A5_16DI_DI_Vars".DI11.cFuncVar)
   END_RUNG
   // the same network as SCL:
   "DIadv"(xInput := "DI12.05.11",
           xInversion := "SS2_A5_16DI_DI_Vars".DI11.xInversion,
           cDelayOffSec := "SS2_A5_16DI_DI_Vars".DI11.cDelayOffSec,
           cDelayOnSec := "SS2_A5_16DI_DI_Vars".DI11.cDelayOnSec,
           xMemoryOut := "SS2_A5_16DI_DI_Vars".DI11.xMemoryOut,
           xMemoryIn := "SS2_A5_16DI_DI_Vars".DI11.xMemoryIn,
           cMemory := "SS2_A5_16DI_DI_Vars".DI11.cMemory,
           iCounterIn := "SS2_A5_16DI_DI_Vars".DI11.iCounterIn,
           iCounterOut := "SS2_A5_16DI_DI_Vars".DI11.iCounterOut,
           xOutputFiltered => "SS2_A5_16DI_DI_Vars".DI11.xOutput,
           xOutputUnFiltered => "SS2_A5_16DI_DI_Vars".DI11.xInput);
   "DIvars"(xInput := "SS2_A5_16DI_DI_Vars".DI11.xOutput,
            iFuncSystem := "SS2_A5_16DI_DI_Vars".DI11.cFuncSystemID,
            iFuncVar := "SS2_A5_16DI_DI_Vars".DI11.cFuncVar);
END_REGION

REGION Network 12: DIb3 / DI01.1.08 EDP під охороною
   RUNG wire#powerrail
      "DIadv"(xInput := wire#w1, xInversion := "SS2_A5_16DI_DI_Vars".DI12.xInversion, cDelayOffSec := "SS2_A5_16DI_DI_Vars".DI12.cDelayOffSec, cDelayOnSec := "SS2_A5_16DI_DI_Vars".DI12.cDelayOnSec, xMemoryOut := "SS2_A5_16DI_DI_Vars".DI12.xMemoryOut, xMemoryIn := "SS2_A5_16DI_DI_Vars".DI12.xMemoryIn, cMemory := "SS2_A5_16DI_DI_Vars".DI12.cMemory, xOutputFiltered => "SS2_A5_16DI_DI_Vars".DI12.xOutput, xOutputUnFiltered => "SS2_A5_16DI_DI_Vars".DI12.xInput, iCounterIn := "SS2_A5_16DI_DI_Vars".DI12.iCounterIn, iCounterOut := "SS2_A5_16DI_DI_Vars".DI12.iCounterOut)
   END_RUNG
   RUNG wire#powerrail
      Contact( "DI12.05.12" )
   END_RUNG wire#w1
   RUNG wire#powerrail
      "DIvars"(xInput := "SS2_A5_16DI_DI_Vars".DI12.xOutput, iFuncSystem := "SS2_A5_16DI_DI_Vars".DI12.cFuncSystemID, iFuncVar := "SS2_A5_16DI_DI_Vars".DI12.cFuncVar)
   END_RUNG
   // the same network as SCL:
   "DIadv"(xInput := "DI12.05.12",
           xInversion := "SS2_A5_16DI_DI_Vars".DI12.xInversion,
           cDelayOffSec := "SS2_A5_16DI_DI_Vars".DI12.cDelayOffSec,
           cDelayOnSec := "SS2_A5_16DI_DI_Vars".DI12.cDelayOnSec,
           xMemoryOut := "SS2_A5_16DI_DI_Vars".DI12.xMemoryOut,
           xMemoryIn := "SS2_A5_16DI_DI_Vars".DI12.xMemoryIn,
           cMemory := "SS2_A5_16DI_DI_Vars".DI12.cMemory,
           iCounterIn := "SS2_A5_16DI_DI_Vars".DI12.iCounterIn,
           iCounterOut := "SS2_A5_16DI_DI_Vars".DI12.iCounterOut,
           xOutputFiltered => "SS2_A5_16DI_DI_Vars".DI12.xOutput,
           xOutputUnFiltered => "SS2_A5_16DI_DI_Vars".DI12.xInput);
   "DIvars"(xInput := "SS2_A5_16DI_DI_Vars".DI12.xOutput,
            iFuncSystem := "SS2_A5_16DI_DI_Vars".DI12.cFuncSystemID,
            iFuncVar := "SS2_A5_16DI_DI_Vars".DI12.cFuncVar);
END_REGION

REGION Network 13: DIb4 / DI01.1.08 EDP під охороною
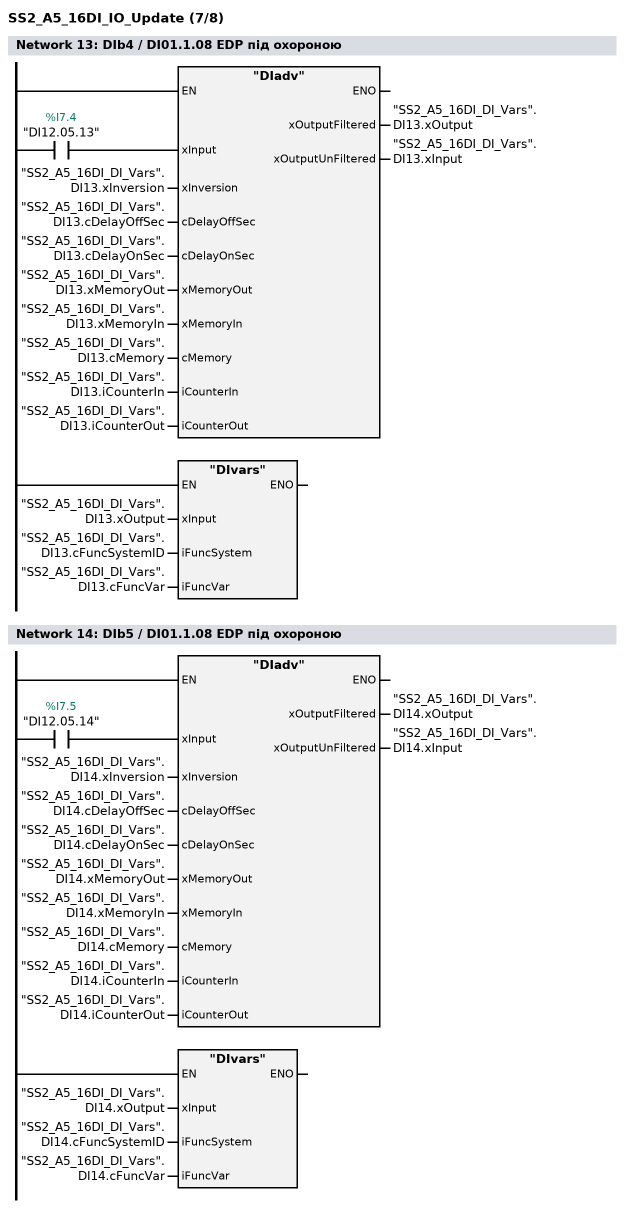
   RUNG wire#powerrail
      "DIadv"(xInput := wire#w1, xInversion := "SS2_A5_16DI_DI_Vars".DI13.xInversion, cDelayOffSec := "SS2_A5_16DI_DI_Vars".DI13.cDelayOffSec, cDelayOnSec := "SS2_A5_16DI_DI_Vars".DI13.cDelayOnSec, xMemoryOut := "SS2_A5_16DI_DI_Vars".DI13.xMemoryOut, xMemoryIn := "SS2_A5_16DI_DI_Vars".DI13.xMemoryIn, cMemory := "SS2_A5_16DI_DI_Vars".DI13.cMemory, xOutputFiltered => "SS2_A5_16DI_DI_Vars".DI13.xOutput, xOutputUnFiltered => "SS2_A5_16DI_DI_Vars".DI13.xInput, iCounterIn := "SS2_A5_16DI_DI_Vars".DI13.iCounterIn, iCounterOut := "SS2_A5_16DI_DI_Vars".DI13.iCounterOut)
   END_RUNG
   RUNG wire#powerrail
      Contact( "DI12.05.13" )
   END_RUNG wire#w1
   RUNG wire#powerrail
      "DIvars"(xInput := "SS2_A5_16DI_DI_Vars".DI13.xOutput, iFuncSystem := "SS2_A5_16DI_DI_Vars".DI13.cFuncSystemID, iFuncVar := "SS2_A5_16DI_DI_Vars".DI13.cFuncVar)
   END_RUNG
   // the same network as SCL:
   "DIadv"(xInput := "DI12.05.13",
           xInversion := "SS2_A5_16DI_DI_Vars".DI13.xInversion,
           cDelayOffSec := "SS2_A5_16DI_DI_Vars".DI13.cDelayOffSec,
           cDelayOnSec := "SS2_A5_16DI_DI_Vars".DI13.cDelayOnSec,
           xMemoryOut := "SS2_A5_16DI_DI_Vars".DI13.xMemoryOut,
           xMemoryIn := "SS2_A5_16DI_DI_Vars".DI13.xMemoryIn,
           cMemory := "SS2_A5_16DI_DI_Vars".DI13.cMemory,
           iCounterIn := "SS2_A5_16DI_DI_Vars".DI13.iCounterIn,
           iCounterOut := "SS2_A5_16DI_DI_Vars".DI13.iCounterOut,
           xOutputFiltered => "SS2_A5_16DI_DI_Vars".DI13.xOutput,
           xOutputUnFiltered => "SS2_A5_16DI_DI_Vars".DI13.xInput);
   "DIvars"(xInput := "SS2_A5_16DI_DI_Vars".DI13.xOutput,
            iFuncSystem := "SS2_A5_16DI_DI_Vars".DI13.cFuncSystemID,
            iFuncVar := "SS2_A5_16DI_DI_Vars".DI13.cFuncVar);
END_REGION

REGION Network 14: DIb5 / DI01.1.08 EDP під охороною
   RUNG wire#powerrail
      "DIadv"(xInput := wire#w1, xInversion := "SS2_A5_16DI_DI_Vars".DI14.xInversion, cDelayOffSec := "SS2_A5_16DI_DI_Vars".DI14.cDelayOffSec, cDelayOnSec := "SS2_A5_16DI_DI_Vars".DI14.cDelayOnSec, xMemoryOut := "SS2_A5_16DI_DI_Vars".DI14.xMemoryOut, xMemoryIn := "SS2_A5_16DI_DI_Vars".DI14.xMemoryIn, cMemory := "SS2_A5_16DI_DI_Vars".DI14.cMemory, xOutputFiltered => "SS2_A5_16DI_DI_Vars".DI14.xOutput, xOutputUnFiltered => "SS2_A5_16DI_DI_Vars".DI14.xInput, iCounterIn := "SS2_A5_16DI_DI_Vars".DI14.iCounterIn, iCounterOut := "SS2_A5_16DI_DI_Vars".DI14.iCounterOut)
   END_RUNG
   RUNG wire#powerrail
      Contact( "DI12.05.14" )
   END_RUNG wire#w1
   RUNG wire#powerrail
      "DIvars"(xInput := "SS2_A5_16DI_DI_Vars".DI14.xOutput, iFuncSystem := "SS2_A5_16DI_DI_Vars".DI14.cFuncSystemID, iFuncVar := "SS2_A5_16DI_DI_Vars".DI14.cFuncVar)
   END_RUNG
   // the same network as SCL:
   "DIadv"(xInput := "DI12.05.14",
           xInversion := "SS2_A5_16DI_DI_Vars".DI14.xInversion,
           cDelayOffSec := "SS2_A5_16DI_DI_Vars".DI14.cDelayOffSec,
           cDelayOnSec := "SS2_A5_16DI_DI_Vars".DI14.cDelayOnSec,
           xMemoryOut := "SS2_A5_16DI_DI_Vars".DI14.xMemoryOut,
           xMemoryIn := "SS2_A5_16DI_DI_Vars".DI14.xMemoryIn,
           cMemory := "SS2_A5_16DI_DI_Vars".DI14.cMemory,
           iCounterIn := "SS2_A5_16DI_DI_Vars".DI14.iCounterIn,
           iCounterOut := "SS2_A5_16DI_DI_Vars".DI14.iCounterOut,
           xOutputFiltered => "SS2_A5_16DI_DI_Vars".DI14.xOutput,
           xOutputUnFiltered => "SS2_A5_16DI_DI_Vars".DI14.xInput);
   "DIvars"(xInput := "SS2_A5_16DI_DI_Vars".DI14.xOutput,
            iFuncSystem := "SS2_A5_16DI_DI_Vars".DI14.cFuncSystemID,
            iFuncVar := "SS2_A5_16DI_DI_Vars".DI14.cFuncVar);
END_REGION

REGION Network 15: DIb6 / DI01.1.08 EDP під охороною
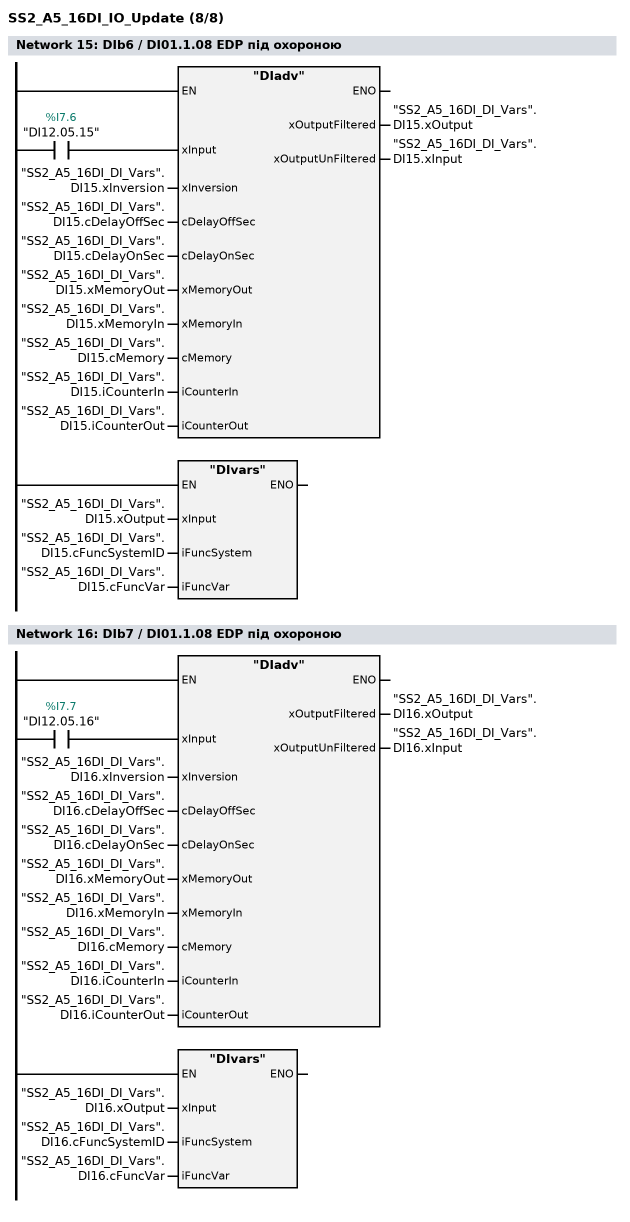
   RUNG wire#powerrail
      "DIadv"(xInput := wire#w1, xInversion := "SS2_A5_16DI_DI_Vars".DI15.xInversion, cDelayOffSec := "SS2_A5_16DI_DI_Vars".DI15.cDelayOffSec, cDelayOnSec := "SS2_A5_16DI_DI_Vars".DI15.cDelayOnSec, xMemoryOut := "SS2_A5_16DI_DI_Vars".DI15.xMemoryOut, xMemoryIn := "SS2_A5_16DI_DI_Vars".DI15.xMemoryIn, cMemory := "SS2_A5_16DI_DI_Vars".DI15.cMemory, xOutputFiltered => "SS2_A5_16DI_DI_Vars".DI15.xOutput, xOutputUnFiltered => "SS2_A5_16DI_DI_Vars".DI15.xInput, iCounterIn := "SS2_A5_16DI_DI_Vars".DI15.iCounterIn, iCounterOut := "SS2_A5_16DI_DI_Vars".DI15.iCounterOut)
   END_RUNG
   RUNG wire#powerrail
      Contact( "DI12.05.15" )
   END_RUNG wire#w1
   RUNG wire#powerrail
      "DIvars"(xInput := "SS2_A5_16DI_DI_Vars".DI15.xOutput, iFuncSystem := "SS2_A5_16DI_DI_Vars".DI15.cFuncSystemID, iFuncVar := "SS2_A5_16DI_DI_Vars".DI15.cFuncVar)
   END_RUNG
   // the same network as SCL:
   "DIadv"(xInput := "DI12.05.15",
           xInversion := "SS2_A5_16DI_DI_Vars".DI15.xInversion,
           cDelayOffSec := "SS2_A5_16DI_DI_Vars".DI15.cDelayOffSec,
           cDelayOnSec := "SS2_A5_16DI_DI_Vars".DI15.cDelayOnSec,
           xMemoryOut := "SS2_A5_16DI_DI_Vars".DI15.xMemoryOut,
           xMemoryIn := "SS2_A5_16DI_DI_Vars".DI15.xMemoryIn,
           cMemory := "SS2_A5_16DI_DI_Vars".DI15.cMemory,
           iCounterIn := "SS2_A5_16DI_DI_Vars".DI15.iCounterIn,
           iCounterOut := "SS2_A5_16DI_DI_Vars".DI15.iCounterOut,
           xOutputFiltered => "SS2_A5_16DI_DI_Vars".DI15.xOutput,
           xOutputUnFiltered => "SS2_A5_16DI_DI_Vars".DI15.xInput);
   "DIvars"(xInput := "SS2_A5_16DI_DI_Vars".DI15.xOutput,
            iFuncSystem := "SS2_A5_16DI_DI_Vars".DI15.cFuncSystemID,
            iFuncVar := "SS2_A5_16DI_DI_Vars".DI15.cFuncVar);
END_REGION

REGION Network 16: DIb7 / DI01.1.08 EDP під охороною
   RUNG wire#powerrail
      "DIadv"(xInput := wire#w1, xInversion := "SS2_A5_16DI_DI_Vars".DI16.xInversion, cDelayOffSec := "SS2_A5_16DI_DI_Vars".DI16.cDelayOffSec, cDelayOnSec := "SS2_A5_16DI_DI_Vars".DI16.cDelayOnSec, xMemoryOut := "SS2_A5_16DI_DI_Vars".DI16.xMemoryOut, xMemoryIn := "SS2_A5_16DI_DI_Vars".DI16.xMemoryIn, cMemory := "SS2_A5_16DI_DI_Vars".DI16.cMemory, xOutputFiltered => "SS2_A5_16DI_DI_Vars".DI16.xOutput, xOutputUnFiltered => "SS2_A5_16DI_DI_Vars".DI16.xInput, iCounterIn := "SS2_A5_16DI_DI_Vars".DI16.iCounterIn, iCounterOut := "SS2_A5_16DI_DI_Vars".DI16.iCounterOut)
   END_RUNG
   RUNG wire#powerrail
      Contact( "DI12.05.16" )
   END_RUNG wire#w1
   RUNG wire#powerrail
      "DIvars"(xInput := "SS2_A5_16DI_DI_Vars".DI16.xOutput, iFuncSystem := "SS2_A5_16DI_DI_Vars".DI16.cFuncSystemID, iFuncVar := "SS2_A5_16DI_DI_Vars".DI16.cFuncVar)
   END_RUNG
   // the same network as SCL:
   "DIadv"(xInput := "DI12.05.16",
           xInversion := "SS2_A5_16DI_DI_Vars".DI16.xInversion,
           cDelayOffSec := "SS2_A5_16DI_DI_Vars".DI16.cDelayOffSec,
           cDelayOnSec := "SS2_A5_16DI_DI_Vars".DI16.cDelayOnSec,
           xMemoryOut := "SS2_A5_16DI_DI_Vars".DI16.xMemoryOut,
           xMemoryIn := "SS2_A5_16DI_DI_Vars".DI16.xMemoryIn,
           cMemory := "SS2_A5_16DI_DI_Vars".DI16.cMemory,
           iCounterIn := "SS2_A5_16DI_DI_Vars".DI16.iCounterIn,
           iCounterOut := "SS2_A5_16DI_DI_Vars".DI16.iCounterOut,
           xOutputFiltered => "SS2_A5_16DI_DI_Vars".DI16.xOutput,
           xOutputUnFiltered => "SS2_A5_16DI_DI_Vars".DI16.xInput);
   "DIvars"(xInput := "SS2_A5_16DI_DI_Vars".DI16.xOutput,
            iFuncSystem := "SS2_A5_16DI_DI_Vars".DI16.cFuncSystemID,
            iFuncVar := "SS2_A5_16DI_DI_Vars".DI16.cFuncVar);
END_REGION
END_FUNCTION

FUNCTION "HVACGeneralParams" : Void   // FC99, LAD
{ S7_Optimized_Access := 'TRUE' }
VERSION : 0.1
// stored: AutoNumber false, IsIECCheckEnabled false, SetENOAutomatically false, UDAEnableTagReadback false
BEGIN

REGION Network 1 (SCL): Season Target
   CASE "HVAC_Vars".Season.cSeasonModeSelection OF
       0:  // Summer;
           "HVAC_Vars".Season.cTarget := 0;
       1:  // Winter
           "HVAC_Vars".Season.cTarget := 1;
       2:  // Midseason
           "HVAC_Vars".Season.cTarget := 2;
       ELSE  // Auto by OAT
           IF "OAT".Temp.rOAT_Actual < "HVAC_Vars".Season.rOATtoWinter THEN
               "HVAC_Vars".Season.cTarget := 1;
           ELSIF "OAT".Temp.rOAT_Actual > "HVAC_Vars".Season.rOATtoSummer THEN
               "HVAC_Vars".Season.cTarget := 0;
           END_IF;
   END_CASE;
END_REGION

REGION Network 2 (SCL): Season Actual
   "HVAC_Vars".Season.cActual := "HVAC_Vars".Season.cTarget;
END_REGION

REGION Network 3: Розклад
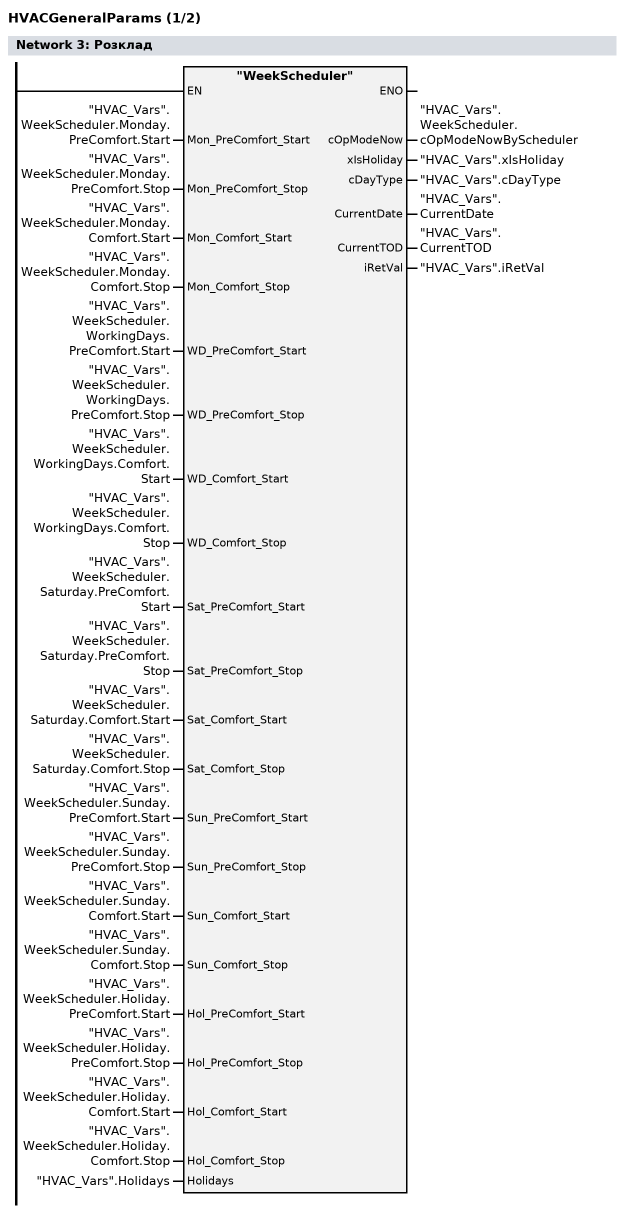
   RUNG wire#powerrail
      "WeekScheduler"(Mon_PreComfort_Start := "HVAC_Vars".WeekScheduler.Monday.PreComfort.Start, Mon_PreComfort_Stop := "HVAC_Vars".WeekScheduler.Monday.PreComfort.Stop, Mon_Comfort_Start := "HVAC_Vars".WeekScheduler.Monday.Comfort.Start, Mon_Comfort_Stop := "HVAC_Vars".WeekScheduler.Monday.Comfort.Stop, WD_PreComfort_Start := "HVAC_Vars".WeekScheduler.WorkingDays.PreComfort.Start, WD_PreComfort_Stop := "HVAC_Vars".WeekScheduler.WorkingDays.PreComfort.Stop, WD_Comfort_Start := "HVAC_Vars".WeekScheduler.WorkingDays.Comfort.Start, WD_Comfort_Stop := "HVAC_Vars".WeekScheduler.WorkingDays.Comfort.Stop, Sat_PreComfort_Start := "HVAC_Vars".WeekScheduler.Saturday.PreComfort.Start, Sat_PreComfort_Stop := "HVAC_Vars".WeekScheduler.Saturday.PreComfort.Stop, Sat_Comfort_Start := "HVAC_Vars".WeekScheduler.Saturday.Comfort.Start, Sat_Comfort_Stop := "HVAC_Vars".WeekScheduler.Saturday.Comfort.Stop, Sun_PreComfort_Start := "HVAC_Vars".WeekScheduler.Sunday.PreComfort.Start, Sun_PreComfort_Stop := "HVAC_Vars".WeekScheduler.Sunday.PreComfort.Stop, Sun_Comfort_Start := "HVAC_Vars".WeekScheduler.Sunday.Comfort.Start, Sun_Comfort_Stop := "HVAC_Vars".WeekScheduler.Sunday.Comfort.Stop, Hol_PreComfort_Start := "HVAC_Vars".WeekScheduler.Holiday.PreComfort.Start, Hol_PreComfort_Stop := "HVAC_Vars".WeekScheduler.Holiday.PreComfort.Stop, Hol_Comfort_Start := "HVAC_Vars".WeekScheduler.Holiday.Comfort.Start, Hol_Comfort_Stop := "HVAC_Vars".WeekScheduler.Holiday.Comfort.Stop, Holidays := "HVAC_Vars".Holidays, cOpModeNow => "HVAC_Vars".WeekScheduler.cOpModeNowByScheduler, xIsHoliday => "HVAC_Vars".xIsHoliday, cDayType => "HVAC_Vars".cDayType, CurrentDate => "HVAC_Vars".CurrentDate, CurrentTOD => "HVAC_Vars".CurrentTOD, iRetVal => "HVAC_Vars".iRetVal)
   END_RUNG
   // the same network as SCL:
   "WeekScheduler"(Mon_PreComfort_Start := "HVAC_Vars".WeekScheduler.Monday.PreComfort.Start,
                   Mon_PreComfort_Stop := "HVAC_Vars".WeekScheduler.Monday.PreComfort.Stop,
                   Mon_Comfort_Start := "HVAC_Vars".WeekScheduler.Monday.Comfort.Start,
                   Mon_Comfort_Stop := "HVAC_Vars".WeekScheduler.Monday.Comfort.Stop,
                   WD_PreComfort_Start := "HVAC_Vars".WeekScheduler.WorkingDays.PreComfort.Start,
                   WD_PreComfort_Stop := "HVAC_Vars".WeekScheduler.WorkingDays.PreComfort.Stop,
                   WD_Comfort_Start := "HVAC_Vars".WeekScheduler.WorkingDays.Comfort.Start,
                   WD_Comfort_Stop := "HVAC_Vars".WeekScheduler.WorkingDays.Comfort.Stop,
                   Sat_PreComfort_Start := "HVAC_Vars".WeekScheduler.Saturday.PreComfort.Start,
                   Sat_PreComfort_Stop := "HVAC_Vars".WeekScheduler.Saturday.PreComfort.Stop,
                   Sat_Comfort_Start := "HVAC_Vars".WeekScheduler.Saturday.Comfort.Start,
                   Sat_Comfort_Stop := "HVAC_Vars".WeekScheduler.Saturday.Comfort.Stop,
                   Sun_PreComfort_Start := "HVAC_Vars".WeekScheduler.Sunday.PreComfort.Start,
                   Sun_PreComfort_Stop := "HVAC_Vars".WeekScheduler.Sunday.PreComfort.Stop,
                   Sun_Comfort_Start := "HVAC_Vars".WeekScheduler.Sunday.Comfort.Start,
                   Sun_Comfort_Stop := "HVAC_Vars".WeekScheduler.Sunday.Comfort.Stop,
                   Hol_PreComfort_Start := "HVAC_Vars".WeekScheduler.Holiday.PreComfort.Start,
                   Hol_PreComfort_Stop := "HVAC_Vars".WeekScheduler.Holiday.PreComfort.Stop,
                   Hol_Comfort_Start := "HVAC_Vars".WeekScheduler.Holiday.Comfort.Start,
                   Hol_Comfort_Stop := "HVAC_Vars".WeekScheduler.Holiday.Comfort.Stop,
                   Holidays := "HVAC_Vars".Holidays,
                   cOpModeNow => "HVAC_Vars".WeekScheduler.cOpModeNowByScheduler,
                   xIsHoliday => "HVAC_Vars".xIsHoliday,
                   cDayType => "HVAC_Vars".cDayType,
                   CurrentDate => "HVAC_Vars".CurrentDate,
                   CurrentTOD => "HVAC_Vars".CurrentTOD,
                   iRetVal => "HVAC_Vars".iRetVal);
END_REGION

REGION Network 4 (SCL): OpMode Target
   CASE "HVAC_Vars".OpModes.cPreselectedOpMode OF
       0:  // Protection;
           "HVAC_Vars".OpModes.cTarget := 0;
       1:  // Economy
           "HVAC_Vars".OpModes.cTarget := 1;
       2:  // PreComf
           "HVAC_Vars".OpModes.cTarget := 2;
       3:  // Comf
           "HVAC_Vars".OpModes.cTarget := 3;
       ELSE  // Auto by Scheduler
           "HVAC_Vars".OpModes.cTarget := "HVAC_Vars".WeekScheduler.cOpModeNowByScheduler;
   END_CASE;
END_REGION

REGION Network 5 (SCL): OpMode Actual
   "HVAC_Vars".OpModes.cActual := "HVAC_Vars".OpModes.cTarget;
END_REGION

REGION Network 6 (SCL): Temp Setpoints to schow on HMI
   CASE "HVAC_Vars".Season.cActual OF
       0:  // Summer
           "HVAC_Vars".RoomTempSetPointforHMI := "HVAC_Vars".SetPoints.Room.Actual.rRATCooling;
       1:  // Winter
           "HVAC_Vars".RoomTempSetPointforHMI := "HVAC_Vars".SetPoints.Room.Actual.rRATHeating;
       ELSE  // Statement section ELSE
           "HVAC_Vars".RoomTempSetPointforHMI := ("HVAC_Vars".SetPoints.Room.Actual.rRATHeating+"HVAC_Vars".SetPoints.Room.Actual.rRATCooling)/2;
   END_CASE;
END_REGION

REGION Network 7 (SCL): Actual OAT
   CASE "OAT".cSelectOATMode OF
       0:
           "OAT".Temp.rOAT_Actual := "HSsAI".AI.rOutdoorTemp_PLC_AI;
       1:
           "OAT".Temp.rOAT_Actual := "OAT".Temp.rOAT_WeatherStation;
       2:
           "OAT".Temp.rOAT_Actual := "OAT".Temp.rOAT_Boilers;
       ELSE  // Statement section ELSE
           "OAT".Temp.rOAT_Actual := "OAT".Temp.rOAT_PLC_IO;
   END_CASE;
END_REGION

REGION Network 8 (SCL): Select values for Actual SP
   CASE "HVAC_Vars".OpModes.cActual OF
       0:  // Protection mode
           "HVAC_Vars".SetPoints.Room.Actual.rRATHeating := "HVAC_Vars".SetPoints.Room.Protection.rRATHeating;
           "HVAC_Vars".SetPoints.Room.Actual.rRATCooling := "HVAC_Vars".SetPoints.Room.Protection.rRATCooling;
           "HVAC_Vars".SetPoints.Room.Actual.rIAQ := "HVAC_Vars".SetPoints.Room.Protection.rIAQ;
           "HVAC_Vars".SetPoints.Room.Actual.rBuildingdP := "HVAC_Vars".SetPoints.Room.Protection.rBuildingdP;
       1:  // Economy mode
           "HVAC_Vars".SetPoints.Room.Actual.rRATHeating := "HVAC_Vars".SetPoints.Room.Econom.rRATHeating;
           "HVAC_Vars".SetPoints.Room.Actual.rRATCooling := "HVAC_Vars".SetPoints.Room.Econom.rRATCooling;
           "HVAC_Vars".SetPoints.Room.Actual.rIAQ := "HVAC_Vars".SetPoints.Room.Econom.rIAQ;
           "HVAC_Vars".SetPoints.Room.Actual.rBuildingdP := "HVAC_Vars".SetPoints.Room.Econom.rBuildingdP;
       2:  // PreComfort mode
           "HVAC_Vars".SetPoints.Room.Actual.rRATHeating := "HVAC_Vars".SetPoints.Room.PreComfort.rRATHeating;
           "HVAC_Vars".SetPoints.Room.Actual.rRATCooling := "HVAC_Vars".SetPoints.Room.PreComfort.rRATCooling;
           "HVAC_Vars".SetPoints.Room.Actual.rIAQ := "HVAC_Vars".SetPoints.Room.PreComfort.rIAQ;
           "HVAC_Vars".SetPoints.Room.Actual.rBuildingdP := "HVAC_Vars".SetPoints.Room.PreComfort.rBuildingdP;
       3:  // Comfort mode
           "HVAC_Vars".SetPoints.Room.Actual.rRATHeating := "HVAC_Vars".SetPoints.Room.Comfort.rRATHeating;
           "HVAC_Vars".SetPoints.Room.Actual.rRATCooling := "HVAC_Vars".SetPoints.Room.Comfort.rRATCooling;
           "HVAC_Vars".SetPoints.Room.Actual.rIAQ := "HVAC_Vars".SetPoints.Room.Comfort.rIAQ;
           "HVAC_Vars".SetPoints.Room.Actual.rBuildingdP := "HVAC_Vars".SetPoints.Room.Comfort.rBuildingdP;
   END_CASE;
END_REGION

REGION Network 9 (SCL)
   //IF "AHUOpModes".OpModes.cActual[#iUnitID] = "AHUOpModes".OpModes.cTarget[#iUnitID] THEN // !!!Змінити на PrevOpMode
   //    // Statement section IF
   //   CASE "AHUOpModes".OpModes.cActual[#iUnitID] OF
   //        0:  // Protection
   //            "AHUSetPoints".SetPoints.Room.Target.RATHeating[#iUnitID] := #rActualStoreSPTempHeating;
   //            "AHUSetPoints".SetPoints.Room.Target.RATCooling[#iUnitID] := #rActualStoreSPTempCooling;
   //            "AHUSetPoints".SetPoints.Room.Target.IAQ[#iUnitID] := #rActualStoreSPIAQ;
   //            "AHUSetPoints".SetPoints.Room.Target.BuildingdP[#iUnitID] := #rActualStoreSPdP;
   //        1:  // Economy
   //            "AHUSetPoints".SetPoints.Room.Target.RATHeating[#iUnitID] := #rEconTempHeating;
   //            "AHUSetPoints".SetPoints.Room.Target.RATCooling[#iUnitID] := #rEconTempCooling;
   //            "AHUSetPoints".SetPoints.Room.Target.IAQ[#iUnitID] := #rEconIAQ;
   //            "AHUSetPoints".SetPoints.Room.Target.BuildingdP[#iUnitID] := #rAHUShiftTempCoolingSP;
   //        2: // Precomfort
   //            "AHUSetPoints".SetPoints.Room.Target.RATHeating[#iUnitID] := #rPreComfTempHeating;
   //            "AHUSetPoints".SetPoints.Room.Target.RATCooling[#iUnitID] := #rPreComfTempCooling;
   //            "AHUSetPoints".SetPoints.Room.Target.IAQ[#iUnitID] := #rPreComfIAQ;
   //            "AHUSetPoints".SetPoints.Room.Target.BuildingdP[#iUnitID] := #rAHUShiftIAQSP;
   //        ELSE  // Statement section ELSE
   //            "AHUSetPoints".SetPoints.Room.Target.RATHeating[#iUnitID] := #rComfTempHeating;
   //            "AHUSetPoints".SetPoints.Room.Target.RATCooling[#iUnitID] := #rComfTempCooling;
   //            "AHUSetPoints".SetPoints.Room.Target.IAQ[#iUnitID] := #rComfIAQ;
   //            "AHUSetPoints".SetPoints.Room.Target.BuildingdP[#iUnitID] := #rAHUShiftdPSP;
   //    END_CASE;
   //    ;
   //END_IF;
END_REGION

REGION Network 10: Weather Depend Calc. Boiler Setpoint
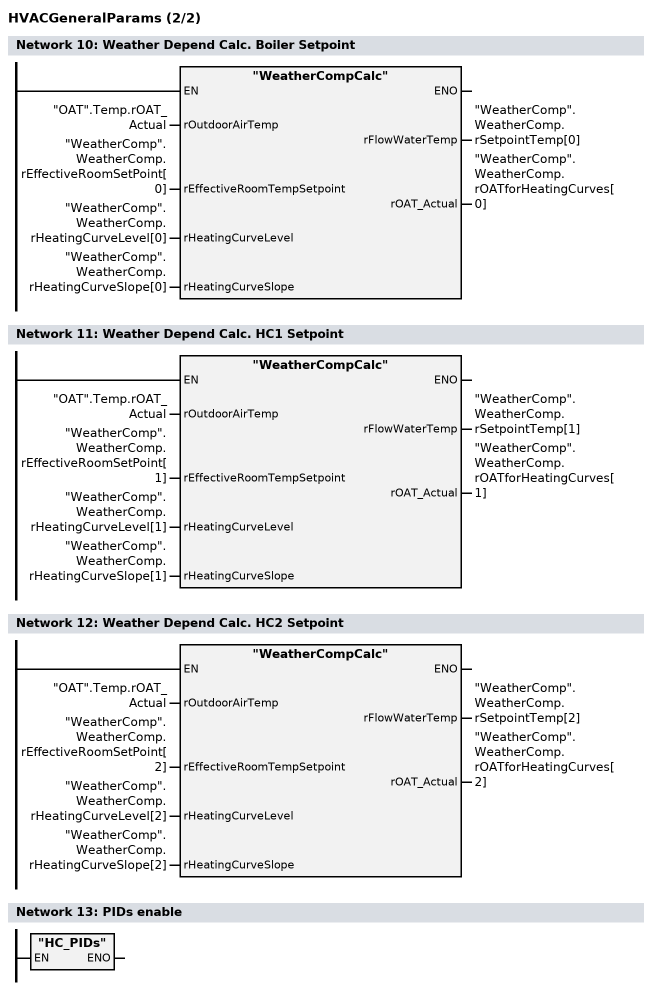
   RUNG wire#powerrail
      "WeatherCompCalc"(rOutdoorAirTemp := "OAT".Temp.rOAT_Actual, rEffectiveRoomTempSetpoint := "WeatherComp".WeatherComp.rEffectiveRoomSetPoint[0], rHeatingCurveLevel := "WeatherComp".WeatherComp.rHeatingCurveLevel[0], rHeatingCurveSlope := "WeatherComp".WeatherComp.rHeatingCurveSlope[0], rFlowWaterTemp => "WeatherComp".WeatherComp.rSetpointTemp[0], rOAT_Actual => "WeatherComp".WeatherComp.rOATforHeatingCurves[0])
   END_RUNG
   // the same network as SCL:
   "WeatherCompCalc"(rOutdoorAirTemp := "OAT".Temp.rOAT_Actual,
                     rEffectiveRoomTempSetpoint := "WeatherComp".WeatherComp.rEffectiveRoomSetPoint[0],
                     rHeatingCurveLevel := "WeatherComp".WeatherComp.rHeatingCurveLevel[0],
                     rHeatingCurveSlope := "WeatherComp".WeatherComp.rHeatingCurveSlope[0],
                     rFlowWaterTemp => "WeatherComp".WeatherComp.rSetpointTemp[0],
                     rOAT_Actual => "WeatherComp".WeatherComp.rOATforHeatingCurves[0]);
END_REGION

REGION Network 11: Weather Depend Calc. HC1 Setpoint
   RUNG wire#powerrail
      "WeatherCompCalc"(rOutdoorAirTemp := "OAT".Temp.rOAT_Actual, rEffectiveRoomTempSetpoint := "WeatherComp".WeatherComp.rEffectiveRoomSetPoint[1], rHeatingCurveLevel := "WeatherComp".WeatherComp.rHeatingCurveLevel[1], rHeatingCurveSlope := "WeatherComp".WeatherComp.rHeatingCurveSlope[1], rFlowWaterTemp => "WeatherComp".WeatherComp.rSetpointTemp[1], rOAT_Actual => "WeatherComp".WeatherComp.rOATforHeatingCurves[1])
   END_RUNG
   // the same network as SCL:
   "WeatherCompCalc"(rOutdoorAirTemp := "OAT".Temp.rOAT_Actual,
                     rEffectiveRoomTempSetpoint := "WeatherComp".WeatherComp.rEffectiveRoomSetPoint[1],
                     rHeatingCurveLevel := "WeatherComp".WeatherComp.rHeatingCurveLevel[1],
                     rHeatingCurveSlope := "WeatherComp".WeatherComp.rHeatingCurveSlope[1],
                     rFlowWaterTemp => "WeatherComp".WeatherComp.rSetpointTemp[1],
                     rOAT_Actual => "WeatherComp".WeatherComp.rOATforHeatingCurves[1]);
END_REGION

REGION Network 12: Weather Depend Calc. HC2 Setpoint
   RUNG wire#powerrail
      "WeatherCompCalc"(rOutdoorAirTemp := "OAT".Temp.rOAT_Actual, rEffectiveRoomTempSetpoint := "WeatherComp".WeatherComp.rEffectiveRoomSetPoint[2], rHeatingCurveLevel := "WeatherComp".WeatherComp.rHeatingCurveLevel[2], rHeatingCurveSlope := "WeatherComp".WeatherComp.rHeatingCurveSlope[2], rFlowWaterTemp => "WeatherComp".WeatherComp.rSetpointTemp[2], rOAT_Actual => "WeatherComp".WeatherComp.rOATforHeatingCurves[2])
   END_RUNG
   // the same network as SCL:
   "WeatherCompCalc"(rOutdoorAirTemp := "OAT".Temp.rOAT_Actual,
                     rEffectiveRoomTempSetpoint := "WeatherComp".WeatherComp.rEffectiveRoomSetPoint[2],
                     rHeatingCurveLevel := "WeatherComp".WeatherComp.rHeatingCurveLevel[2],
                     rHeatingCurveSlope := "WeatherComp".WeatherComp.rHeatingCurveSlope[2],
                     rFlowWaterTemp => "WeatherComp".WeatherComp.rSetpointTemp[2],
                     rOAT_Actual => "WeatherComp".WeatherComp.rOATforHeatingCurves[2]);
END_REGION

REGION Network 13: PIDs enable
   RUNG wire#powerrail
      "HC_PIDs"()
   END_RUNG
   // the same network as SCL:
   "HC_PIDs"();
END_REGION
END_FUNCTION

FUNCTION "WeekScheduler" : Void   // FC98, LAD
{ S7_Optimized_Access := 'TRUE' }
VERSION : 0.1
// stored: AutoNumber false, IsIECCheckEnabled false, SetENOAutomatically false, UDAEnableTagReadback false
   VAR_INPUT
      Mon_PreComfort_Start : Time_Of_Day;
      Mon_PreComfort_Stop : Time_Of_Day;
      Mon_Comfort_Start : Time_Of_Day;
      Mon_Comfort_Stop : Time_Of_Day;
      WD_PreComfort_Start : Time_Of_Day;
      WD_PreComfort_Stop : Time_Of_Day;
      WD_Comfort_Start : Time_Of_Day;
      WD_Comfort_Stop : Time_Of_Day;
      Sat_PreComfort_Start : Time_Of_Day;
      Sat_PreComfort_Stop : Time_Of_Day;
      Sat_Comfort_Start : Time_Of_Day;
      Sat_Comfort_Stop : Time_Of_Day;
      Sun_PreComfort_Start : Time_Of_Day;
      Sun_PreComfort_Stop : Time_Of_Day;
      Sun_Comfort_Start : Time_Of_Day;
      Sun_Comfort_Stop : Time_Of_Day;
      Hol_PreComfort_Start : Time_Of_Day;
      Hol_PreComfort_Stop : Time_Of_Day;
      Hol_Comfort_Start : Time_Of_Day;
      Hol_Comfort_Stop : Time_Of_Day;
      Holidays : Array[1..4] of Date;
   END_VAR
   VAR_OUTPUT
      cOpModeNow : Byte;
      xIsHoliday : Bool;
      cDayType : Byte;   // 1-WD/2-Sat/3-Sun/4 - Hol
      CurrentDate : Date;
      CurrentTOD : Time_Of_Day;
      iRetVal : Int;
   END_VAR
   VAR_TEMP
      NowDTL : DTL;
      i : Int;
      PreComfStart : Time_Of_Day;
      PreComfStop : Time_Of_Day;
      ComfStart : Time_Of_Day;
      ComfStop : Time_Of_Day;
      xInPreComf : Bool;
      xInComf : Bool;
   END_VAR
BEGIN

REGION Network 1 (SCL): // Значення за замовчуванням
       // Значення за замовчуванням
      // #cOpModeNow := 1; // Економ
      // #xIsHoliday := FALSE;
      // #cDayType := 1; // Робочий
      // #CurrentDate := DATE#1990-01-01;
      // #CurrentTOD := TOD#00:00:00;
      // #iRetVal := 0;
END_REGION

REGION Network 2 (SCL): Час на CPU
   // Читаємо локальний час CPU
   #iRetVal := RD_LOC_T(OUT => #NowDTL);

   // Якщо час не прочитався - лишаємо Економ
   //IF #iRetVal >= 16#8000 THEN
   //    #cOpModeNow := 1;
   //    RETURN;
   //END_IF;

   // Виділяємо дату і час
   #CurrentDate := DTL_TO_DATE(#NowDTL);
   #CurrentTOD := DTL_TO_TOD(#NowDTL);
END_REGION

REGION Network 3 (SCL): // Перевірка святкового дня
   // Перевірка святкового дня
   FOR #i := 1 TO 3 DO
       IF #Holidays[#i] = #CurrentDate THEN
           #xIsHoliday := TRUE;
           EXIT;
       END_IF;
   END_FOR;
END_REGION

REGION Network 4 (SCL): 0-WD/1-Mon/2-Sat/3-Sun/4 - Hol
       // Визначення типу дня
       IF #xIsHoliday THEN
           #cDayType := 4; // Святковий
       ELSE
           // Weekday: 1=Sunday ... 7=Saturday
           CASE #NowDTL.WEEKDAY OF
               7:
                   #cDayType := 2; // Субота
               1:
                   #cDayType := 3; // Неділя
               2:
                   #cDayType := 1; // Понеділок
               ELSE
                   #cDayType := 0; // Робочий
           END_CASE;
       END_IF;
END_REGION

REGION Network 5 (SCL): // Вибір активного розкладу
   // Вибір активного розкладу
   CASE #cDayType OF
       0: // Робочий
           #PreComfStart := #WD_PreComfort_Start;
           #PreComfStop := #WD_PreComfort_Stop;
           #ComfStart := #WD_Comfort_Start;
           #ComfStop := #WD_Comfort_Stop;

       1: // Понеділок
           #PreComfStart := #Mon_PreComfort_Start;
           #PreComfStop := #Mon_PreComfort_Stop;
           #ComfStart := #Mon_Comfort_Start;
           #ComfStop := #Mon_Comfort_Stop;

       2: // Субота
           #PreComfStart := #Sat_PreComfort_Start;
           #PreComfStop := #Sat_PreComfort_Stop;
           #ComfStart := #Sat_Comfort_Start;
           #ComfStop := #Sat_Comfort_Stop;

       3: // Неділя
           #PreComfStart := #Sun_PreComfort_Start;
           #PreComfStop := #Sun_PreComfort_Stop;
           #ComfStart := #Sun_Comfort_Start;
           #ComfStop := #Sun_Comfort_Stop;

       4: // Святковий
           #PreComfStart := #Hol_PreComfort_Start;
           #PreComfStop := #Hol_PreComfort_Stop;
           #ComfStart := #Hol_Comfort_Start;
           #ComfStop := #Hol_Comfort_Stop;

       ELSE
           #PreComfStart := TOD#00:00:00;
           #PreComfStop := TOD#00:00:00;
           #ComfStart := TOD#00:00:00;
           #ComfStop := TOD#00:00:00;

   END_CASE;
END_REGION

REGION Network 6 (SCL): // Перевірка потрапляння в інтервали InComf
       IF #ComfStart = #ComfStop THEN
           // трактуємо як "вікно вимкнене"
           #xInComf := FALSE;

       ELSIF #ComfStart <  #ComfStop THEN
           // звичайний інтервал, наприклад 06:00..22:00
           #xInComf := (#CurrentTOD >= #ComfStart) AND (#CurrentTOD < #ComfStop);

       ELSE
           // інтервал через північ, наприклад 22:00..06:00
           //#xInComf := (#CurrentTOD >= #ComfStart) OR (#CurrentTOD < #ComfStop);
           #xInComf := FALSE;
       END_IF;
END_REGION

REGION Network 7 (SCL): // Перевірка потрапляння в інтервали InPreComf
       IF #PreComfStart = #PreComfStop THEN
           // трактуємо як "вікно вимкнене"
           #xInPreComf := FALSE;

       ELSIF #PreComfStart < #PreComfStop THEN
           // звичайний інтервал, наприклад 06:00..22:00
           #xInPreComf := (#CurrentTOD >= #PreComfStart) AND (#CurrentTOD < #PreComfStop);

       ELSE
           // інтервал через північ, наприклад 22:00..06:00
           //#xInComf := (#CurrentTOD >= #ComfStart) OR (#CurrentTOD < #ComfStop);
           #xInPreComf := FALSE;
       END_IF;
END_REGION

REGION Network 8 (SCL): // Пріоритет: Комфорт > Прекомфорт > Економ
       // Пріоритет: Комфорт > Прекомфорт > Економ
       IF #xInComf THEN
           #cOpModeNow := 3; // Комфорт
       ELSIF #xInPreComf THEN
           #cOpModeNow := 2; // Прекомфорт
       ELSE
           #cOpModeNow := 1; // Економ
       END_IF;
END_REGION
END_FUNCTION

FUNCTION "WeatherCompCalc" : Void
{ S7_Optimized_Access := 'TRUE' }
VERSION : 0.1
   VAR_INPUT 
      rOutdoorAirTemp : Real;
      rEffectiveRoomTempSetpoint : Real;
      rHeatingCurveLevel : Real;
      rHeatingCurveSlope : Real;
   END_VAR

   VAR_OUTPUT 
      rFlowWaterTemp : Real;
      rOAT_Actual : Real;
   END_VAR

   VAR_TEMP 
      rTemp : Real;
   END_VAR


BEGIN
	IF (#rEffectiveRoomTempSetpoint > #rOutdoorAirTemp) THEN
	    #rTemp := #rEffectiveRoomTempSetpoint + #rHeatingCurveSlope * 1.91 * EXP(0.816 * LN(#rEffectiveRoomTempSetpoint - #rOutdoorAirTemp)) + #rHeatingCurveLevel;
	ELSE
	    #rTemp := #rEffectiveRoomTempSetpoint;
	END_IF;
	
	IF #rTemp > 90 THEN
	    #rFlowWaterTemp := 90;
	ELSIF #rTemp < #rEffectiveRoomTempSetpoint THEN
	    #rFlowWaterTemp := #rEffectiveRoomTempSetpoint;
	ELSE
	    #rFlowWaterTemp := #rTemp;
	END_IF;
	
	#rOAT_Actual := #rOutdoorAirTemp;
END_FUNCTION

FUNCTION "HC_PIDs" : Void   // FC1019, LAD
{ S7_Optimized_Access := 'TRUE' }
VERSION : 0.1
// stored: AutoNumber false, IsIECCheckEnabled false, SetENOAutomatically false, UDAEnableTagReadback false
BEGIN

REGION Network 1
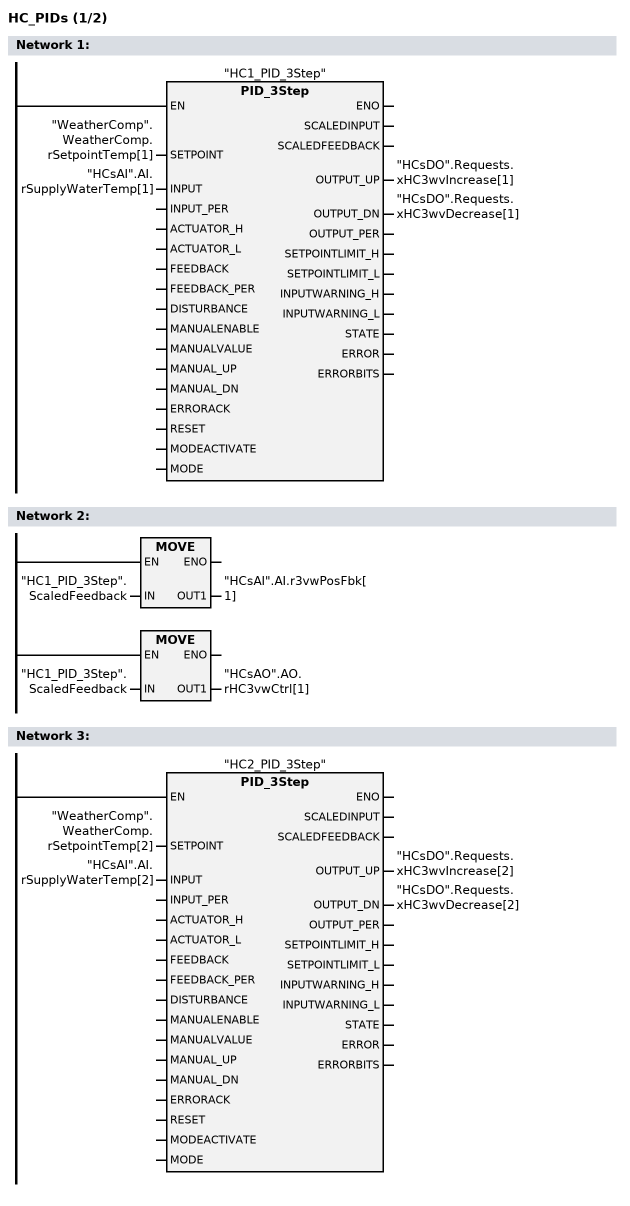
   RUNG wire#powerrail
      "HC1_PID_3Step".PID_3Step(Setpoint := "WeatherComp".WeatherComp.rSetpointTemp[1], Input := "HCsAI".AI.rSupplyWaterTemp[1], Input_PER :=, Actuator_H :=, Actuator_L :=, Feedback :=, Feedback_PER :=, Disturbance :=, ManualEnable :=, ManualValue :=, Manual_UP :=, Manual_DN :=, ErrorAck :=, Reset :=, ModeActivate :=, Mode :=, ScaledInput =>, ScaledFeedback =>, Output_UP => "HCsDO".Requests.xHC3wvIncrease[1], Output_DN => "HCsDO".Requests.xHC3wvDecrease[1], Output_PER =>, SetpointLimit_H =>, SetpointLimit_L =>, InputWarning_H =>, InputWarning_L =>, State =>, Error =>, ErrorBits =>)
   END_RUNG
   // the same network as SCL:
   "HC1_PID_3Step"(Setpoint := "WeatherComp".WeatherComp.rSetpointTemp[1],   // PID_3Step
                   Input := "HCsAI".AI.rSupplyWaterTemp[1],
                   Output_UP => "HCsDO".Requests.xHC3wvIncrease[1],
                   Output_DN => "HCsDO".Requests.xHC3wvDecrease[1]);
END_REGION

REGION Network 2
   RUNG wire#powerrail
      Move(in := "HC1_PID_3Step".ScaledFeedback, out1 => "HCsAI".AI.r3vwPosFbk[1])
   END_RUNG
   RUNG wire#powerrail
      Move(in := "HC1_PID_3Step".ScaledFeedback, out1 => "HCsAO".AO.rHC3vwCtrl[1])
   END_RUNG
   // the same network as SCL:
   "HCsAI".AI.r3vwPosFbk[1] := "HC1_PID_3Step".ScaledFeedback;
   "HCsAO".AO.rHC3vwCtrl[1] := "HC1_PID_3Step".ScaledFeedback;
END_REGION

REGION Network 3
   RUNG wire#powerrail
      "HC2_PID_3Step".PID_3Step(Setpoint := "WeatherComp".WeatherComp.rSetpointTemp[2], Input := "HCsAI".AI.rSupplyWaterTemp[2], Input_PER :=, Actuator_H :=, Actuator_L :=, Feedback :=, Feedback_PER :=, Disturbance :=, ManualEnable :=, ManualValue :=, Manual_UP :=, Manual_DN :=, ErrorAck :=, Reset :=, ModeActivate :=, Mode :=, ScaledInput =>, ScaledFeedback =>, Output_UP => "HCsDO".Requests.xHC3wvIncrease[2], Output_DN => "HCsDO".Requests.xHC3wvDecrease[2], Output_PER =>, SetpointLimit_H =>, SetpointLimit_L =>, InputWarning_H =>, InputWarning_L =>, State =>, Error =>, ErrorBits =>)
   END_RUNG
   // the same network as SCL:
   "HC2_PID_3Step"(Setpoint := "WeatherComp".WeatherComp.rSetpointTemp[2],   // PID_3Step
                   Input := "HCsAI".AI.rSupplyWaterTemp[2],
                   Output_UP => "HCsDO".Requests.xHC3wvIncrease[2],
                   Output_DN => "HCsDO".Requests.xHC3wvDecrease[2]);
END_REGION

REGION Network 4
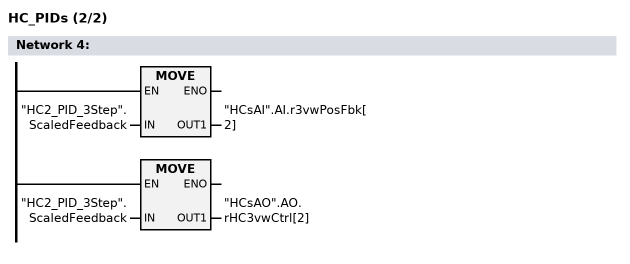
   RUNG wire#powerrail
      Move(in := "HC2_PID_3Step".ScaledFeedback, out1 => "HCsAI".AI.r3vwPosFbk[2])
   END_RUNG
   RUNG wire#powerrail
      Move(in := "HC2_PID_3Step".ScaledFeedback, out1 => "HCsAO".AO.rHC3vwCtrl[2])
   END_RUNG
   // the same network as SCL:
   "HCsAI".AI.r3vwPosFbk[2] := "HC2_PID_3Step".ScaledFeedback;
   "HCsAO".AO.rHC3vwCtrl[2] := "HC2_PID_3Step".ScaledFeedback;
END_REGION
END_FUNCTION

FUNCTION "AHU_Main" : Void   // FC100, FBD
{ S7_Optimized_Access := 'TRUE' }
VERSION : 0.1
// stored: AutoNumber false, IsIECCheckEnabled false, SetENOAutomatically false, UDAEnableTagReadback false
   VAR_INPUT
      iUnitID : Int;   // 1=AHUFood, 2=AHUNonFood
   END_VAR
   VAR_TEMP
      FA_temp : Real;
   END_VAR
BEGIN

REGION Network 1 (SCL): Actual Room (salles area temp)
   // 0=PLC_IO, 1=LoraAvg, 2=MSensor,3 =PLC
   CASE "AHUAI".AI.cRoomTempSelect[#iUnitID] OF
       0:  // 
           "AHUAI".AI.rRoomAirTemp_Actual[#iUnitID] := "AHUAI".AI.rRoomAirTemp_PLC_AI[#iUnitID];
       1:  // 
           "AHUAI".AI.rRoomAirTemp_Actual[#iUnitID] := "AHUAI".AI.rRoomAirTemp_LoraAvg[#iUnitID];
       2: // 
           "AHUAI".AI.rRoomAirTemp_Actual[#iUnitID] := "AHUAI".AI.rRoomAirTemp_MSensor[#iUnitID];
       ELSE
           "AHUAI".AI.rRoomAirTemp_Actual[#iUnitID] := "AHUAI".AI.rRoomAirTemp_PLC_AI[#iUnitID];
   END_CASE;
END_REGION

REGION Network 2
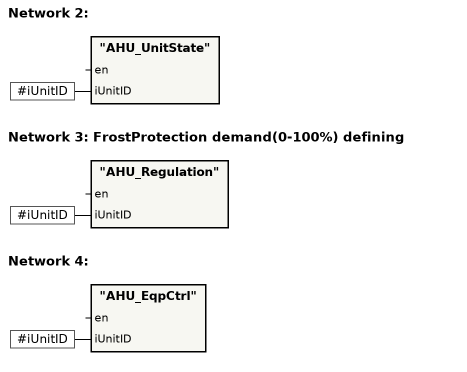
   "AHU_UnitState"(iUnitID := #iUnitID);
END_REGION

REGION Network 3: FrostProtection demand(0-100%) defining
   "AHU_Regulation"(iUnitID := #iUnitID);
END_REGION

REGION Network 4
   "AHU_EqpCtrl"(iUnitID := #iUnitID);
END_REGION
END_FUNCTION

FUNCTION "AHU_UnitState" : Void   // FC60100, FBD
{ S7_Optimized_Access := 'TRUE' }
VERSION : 0.1
// stored: AutoNumber false, IsIECCheckEnabled false, SetENOAutomatically false, UDAEnableTagReadback false
   VAR_INPUT
      iUnitID : Int;   // 1=AHUFood, 2=AHUNonFood
   END_VAR
   VAR_TEMP
      FA_temp : Real;
   END_VAR
BEGIN

REGION Network 1 (SCL)
   IF "FirstScan" THEN
       ;
       "AHUUnitStates".UnitStates.cActual[#iUnitID] := 0;
       "AHUUnitStates".UnitStates.cTarget[#iUnitID] := 0;
   END_IF;
END_REGION

REGION Network 2: AHUs Actual Operation Mode define
   // Operation Modes                                                 Unit State
   // 0=Protection                                                         0=Stopped
   // 1=Economy                                                           1=Checking-up  
   // 2=PreComfort                                                       2=Preheating
   // 3=Comfor                                                              3=Starting 
   // 4=Auto(Scheduler)                                              4=RecirculatingOperation (Protection)
   //                                                                                 5=Sustained Mode (Economy setpoints)
   //                                                                                 6=Sustained Mode (PreComfort setpoints) 
   //                                                                                 7=Comfort  operation
   //                                                                                 8=Stopping
   //                                                                                 9=Blocking
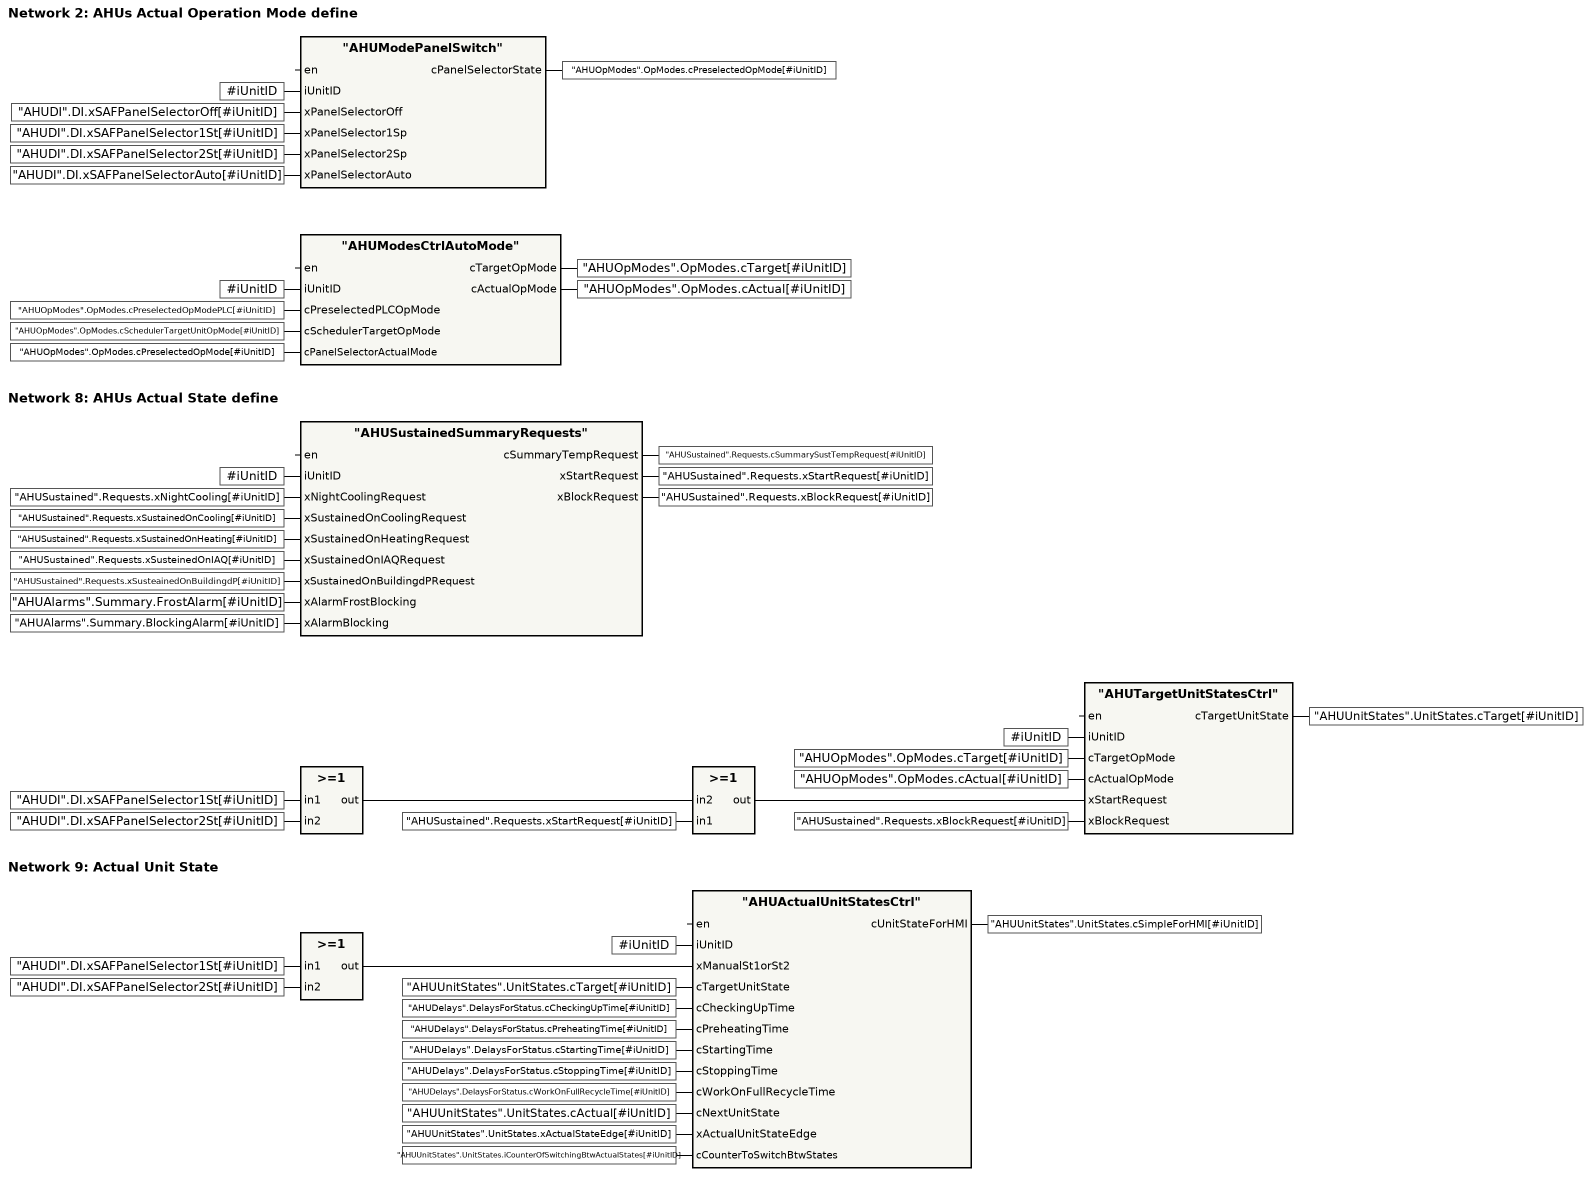
   "AHUModePanelSwitch"(iUnitID := #iUnitID,
                        xPanelSelectorOff := "AHUDI".DI.xSAFPanelSelectorOff[#iUnitID],
                        xPanelSelector1Sp := "AHUDI".DI.xSAFPanelSelector1St[#iUnitID],
                        xPanelSelector2Sp := "AHUDI".DI.xSAFPanelSelector2St[#iUnitID],
                        xPanelSelectorAuto := "AHUDI".DI.xSAFPanelSelectorAuto[#iUnitID],
                        cPanelSelectorState => "AHUOpModes".OpModes.cPreselectedOpMode[#iUnitID]);
   "AHUModesCtrlAutoMode"(iUnitID := #iUnitID,
                          cPreselectedPLCOpMode := "AHUOpModes".OpModes.cPreselectedOpModePLC[#iUnitID],
                          cSchedulerTargetOpMode := "AHUOpModes".OpModes.cSchedulerTargetUnitOpMode[#iUnitID],
                          cPanelSelectorActualMode := "AHUOpModes".OpModes.cPreselectedOpMode[#iUnitID],
                          cTargetOpMode => "AHUOpModes".OpModes.cTarget[#iUnitID],
                          cActualOpMode => "AHUOpModes".OpModes.cActual[#iUnitID]);
END_REGION

REGION Network 3 (SCL): NightCooling Request
   IF FALSE THEN
       // Statement section IF
       "AHUSustained".Requests.xNightCooling[#iUnitID] := TRUE;
   ELSE
       "AHUSustained".Requests.xNightCooling[#iUnitID] := FALSE;
   END_IF;
END_REGION

REGION Network 4 (SCL): Sustained requests cooling
   IF "AHURegulators".Regulators.State.cTempCooling[#iUnitID] > 0 THEN
       // Statement section IF
       ;
   ELSE
       "AHUSustained".Requests.xSustainedOnCooling[#iUnitID] := FALSE;
   END_IF;
END_REGION

REGION Network 5 (SCL): Sustained request heating
   IF "AHURegulators".Regulators.State.cTempHeating[#iUnitID] > 0 THEN
       // Statement section IF
       ;
   ELSE
       "AHUSustained".Requests.xSustainedOnHeating[#iUnitID] := FALSE;
   END_IF;
END_REGION

REGION Network 6 (SCL): Sustained request IAQ
   IF "AHURegulators".Regulators.State.cIAQ[#iUnitID] > 0 THEN
       // Statement section IF
       ;
   ELSE
       "AHUSustained".Requests.xSusteinedOnIAQ[#iUnitID] := FALSE;
   END_IF;
END_REGION

REGION Network 7 (SCL): Sustained request Building Pressurisation
   IF "AHURegulators".Regulators.State.cBuildingdP[#iUnitID] > 0 THEN
       // Statement section IF
       ;
   ELSE
       "AHUSustained".Requests.xSusteainedOnBuildingdP[#iUnitID] := FALSE;
   END_IF;
END_REGION

REGION Network 8: AHUs Actual State define
   // Operation Modes                                                 Unit State
   // 0=Protection                                                         0=Stopped
   // 1=Economy                                                           1=Checking-up  
   // 2=PreComfort                                                       2=Preheating
   // 3=Comfor                                                              3=Starting 
   // 4=Auto(Scheduler)                                              4=RecirculatingOperation
   //                                                                                 5=Sustained Mode (Economy setpoints)
   //                                                                                 6=Sustained Mode (PreComfort setpoints) 
   //                                                                                 7=Comfort  operation
   //                                                                                 8=Stopping
   //                                                                                 9=Blocking
   "AHUSustainedSummaryRequests"(iUnitID := #iUnitID,
                           xNightCoolingRequest := "AHUSustained".Requests.xNightCooling[#iUnitID],
                           xSustainedOnCoolingRequest := "AHUSustained".Requests.xSustainedOnCooling[#iUnitID],
                           xSustainedOnHeatingRequest := "AHUSustained".Requests.xSustainedOnHeating[#iUnitID],
                           xSustainedOnIAQRequest := "AHUSustained".Requests.xSusteinedOnIAQ[#iUnitID],
                           xSustainedOnBuildingdPRequest := "AHUSustained".Requests.xSusteainedOnBuildingdP[#iUnitID],
                           xAlarmFrostBlocking := "AHUAlarms".Summary.FrostAlarm[#iUnitID],
                           xAlarmBlocking := "AHUAlarms".Summary.BlockingAlarm[#iUnitID],
                           cSummaryTempRequest => "AHUSustained".Requests.cSummarySustTempRequest[#iUnitID],
                           xStartRequest => "AHUSustained".Requests.xStartRequest[#iUnitID],
                           xBlockRequest => "AHUSustained".Requests.xBlockRequest[#iUnitID]);
   "AHUTargetUnitStatesCtrl"(iUnitID := #iUnitID,
                           cTargetOpMode := "AHUOpModes".OpModes.cTarget[#iUnitID],
                           cActualOpMode := "AHUOpModes".OpModes.cActual[#iUnitID],
                           xStartRequest := "AHUDI".DI.xSAFPanelSelector1St[#iUnitID] OR "AHUDI".DI.xSAFPanelSelector2St[#iUnitID] OR "AHUSustained".Requests.xStartRequest[#iUnitID],
                           xBlockRequest := "AHUSustained".Requests.xBlockRequest[#iUnitID],
                           cTargetUnitState => "AHUUnitStates".UnitStates.cTarget[#iUnitID]);
END_REGION

REGION Network 9: Actual Unit State
   "AHUActualUnitStatesCtrl"(iUnitID := #iUnitID,
                           xManualSt1orSt2 := "AHUDI".DI.xSAFPanelSelector1St[#iUnitID] OR "AHUDI".DI.xSAFPanelSelector2St[#iUnitID],
                           cTargetUnitState := "AHUUnitStates".UnitStates.cTarget[#iUnitID],
                           cCheckingUpTime := "AHUDelays".DelaysForStatus.cCheckingUpTime[#iUnitID],
                           cPreheatingTime := "AHUDelays".DelaysForStatus.cPreheatingTime[#iUnitID],
                           cStartingTime := "AHUDelays".DelaysForStatus.cStartingTime[#iUnitID],
                           cStoppingTime := "AHUDelays".DelaysForStatus.cStoppingTime[#iUnitID],
                           cWorkOnFullRecycleTime := "AHUDelays".DelaysForStatus.cWorkOnFullRecycleTime[#iUnitID],
                           cNextUnitState := "AHUUnitStates".UnitStates.cActual[#iUnitID],
                           xActualUnitStateEdge := "AHUUnitStates".UnitStates.xActualStateEdge[#iUnitID],
                           cCounterToSwitchBtwStates := "AHUUnitStates".UnitStates.iCounterOfSwitchingBtwActualStates[#iUnitID],
                           cUnitStateForHMI => "AHUUnitStates".UnitStates.cSimpleForHMI[#iUnitID]);
END_REGION
END_FUNCTION

FUNCTION "AHUModePanelSwitch" : Void   // FC60101, LAD
{ S7_Optimized_Access := 'TRUE' }
VERSION : 0.1
// stored: AutoNumber false, IsIECCheckEnabled false, SetENOAutomatically false, UDAEnableTagReadback false
   VAR_INPUT
      iUnitID : Int;
      xPanelSelectorOff : Bool;
      xPanelSelector1Sp : Bool;
      xPanelSelector2Sp : Bool;
      xPanelSelectorAuto : Bool;
   END_VAR
   VAR_OUTPUT
      cPanelSelectorState : Byte;
   END_VAR
BEGIN

REGION Network 1 (SCL)
   IF #xPanelSelectorOff THEN
       #cPanelSelectorState := 0;//Off
   ELSIF #xPanelSelector1Sp THEN
       #cPanelSelectorState := 2;//Speed1
   ELSIF #xPanelSelector2Sp THEN
       #cPanelSelectorState := 3;//Speed2
   ELSE
       #cPanelSelectorState := 4;//Auto
   END_IF;
END_REGION
END_FUNCTION

FUNCTION "AHUModesCtrlAutoMode" : Void   // FC60102, LAD
{ S7_Optimized_Access := 'TRUE' }
VERSION : 0.1
// stored: AutoNumber false, IsIECCheckEnabled false, SetENOAutomatically false, UDAEnableTagReadback false
   VAR_INPUT
      iUnitID : Int;
      cPreselectedPLCOpMode : Byte;
      cSchedulerTargetOpMode : Byte;
      cPanelSelectorActualMode : Byte;
   END_VAR
   VAR_OUTPUT
      cTargetOpMode : Byte;
      cActualOpMode : Byte;
   END_VAR
   VAR_TEMP
      TargetUnitMode_old : Int;
      ResetActualOperationMode : Bool;
   END_VAR
BEGIN

REGION Network 1 (SCL)
   CASE #cPanelSelectorActualMode OF
       0:                                                     // Switch is in OFF
           #cTargetOpMode := 0;                               //Protection
       1:
           ;
       2:                                                     // Switch is in Sp1
           #cTargetOpMode := 2;                               //Precomfort     ;
       3:                                                     // Switch is in Sp2
           #cTargetOpMode := 3;                               //Precomfort     ;
       ELSE                                                   // Switch is in Auto
           IF #cPreselectedPLCOpMode = 4 THEN                 // PLC mode 3=Scheduler
               #cTargetOpMode := #cSchedulerTargetOpMode;     // 
           ELSE                                               //mode-0-1-2-
               #cTargetOpMode := #cPreselectedPLCOpMode;
           END_IF;
   END_CASE;
END_REGION

REGION Network 2 (SCL)
   IF #cTargetOpMode <> #cActualOpMode THEN
       // Update Actual OP Mode
       #cActualOpMode := #cTargetOpMode;
   END_IF;
END_REGION

REGION Network 3 (SCL)
   IF #cActualOpMode <> "cActualOpModePrevOne" THEN
       "iActualOpModeCounter" := "iActualOpModeCounter" + 1;
   END_IF;

   "cActualOpModePrevOne" := #cActualOpMode;
END_REGION
END_FUNCTION

FUNCTION "AHUSustainedSummaryRequests" : Void   // FC60103, LAD
{ S7_Optimized_Access := 'TRUE' }
VERSION : 0.1
// stored: AutoNumber false, IsIECCheckEnabled false, SetENOAutomatically false, UDAEnableTagReadback false
   VAR_INPUT
      iUnitID : Int;
      xNightCoolingRequest : Bool;
      xSustainedOnCoolingRequest : Bool;
      xSustainedOnHeatingRequest : Bool;
      xSustainedOnIAQRequest : Bool;
      xSustainedOnBuildingdPRequest : Bool;
      xAlarmFrostBlocking : Bool;
      xAlarmBlocking : Bool;
   END_VAR
   VAR_OUTPUT
      cSummaryTempRequest : Byte;
      xStartRequest : Bool;
      xBlockRequest : Bool;
   END_VAR
BEGIN

REGION Network 1 (SCL)
   #xStartRequest := #xNightCoolingRequest OR
   #xSustainedOnCoolingRequest OR
   #xSustainedOnHeatingRequest OR  
   #xSustainedOnIAQRequest OR
   #xSustainedOnBuildingdPRequest;
END_REGION

REGION Network 2 (SCL)
   #xBlockRequest := #xAlarmFrostBlocking OR
   #xAlarmBlocking;
END_REGION

REGION Network 3 (SCL)
   IF #xNightCoolingRequest THEN
       #cSummaryTempRequest := 3;
   ELSIF #xSustainedOnCoolingRequest THEN
       #cSummaryTempRequest := 2;
   ELSE
       IF #xSustainedOnHeatingRequest THEN
           #cSummaryTempRequest := 1;
       ELSE
           #cSummaryTempRequest := 0;
       END_IF;

   END_IF;
END_REGION
END_FUNCTION

FUNCTION "AHUTargetUnitStatesCtrl" : Void   // FC60104, LAD
{ S7_Optimized_Access := 'TRUE' }
VERSION : 0.1
// Operation Modes                                                 Unit State
// 0=Protection                                                         0=Stopped
// 1=Economy                                                           1=Checking-up  
// 2=PreComfort                                                       2=Preheating
// 3=Comfor                                                              3=Starting 
// 4=Auto(Scheduler)                                              4=RecirculatingOperation
//                                                                                 5=Economy Operation                                                                                                                                            6=PreComfort Operation 
//                                                                                 7=Comfort  operation
//                                                                                 8=Stopping
//                                                                                 9=Blocking
// stored: AutoNumber false, IsIECCheckEnabled false, SetENOAutomatically false, UDAEnableTagReadback false
   VAR_INPUT
      iUnitID : Int;
      cTargetOpMode : Byte;
      cActualOpMode : Byte;
      xStartRequest : Bool;
      xBlockRequest : Bool;
   END_VAR
   VAR_OUTPUT
      cTargetUnitState : Byte;
   END_VAR
BEGIN

REGION Network 1 (SCL)
   CASE #cActualOpMode OF
       0:                                                  // OpMode is OFF(Protection)
           IF #xBlockRequest THEN                               // Stop by alarm      
               #cTargetUnitState := 9;
           ELSE 
               #cTargetUnitState := 0;
           END_IF;
       1:                                                  // Economy mode 
           IF #xBlockRequest THEN                               // Stop by alarm      
               #cTargetUnitState := 9;
           ELSIF #xStartRequest THEN                           //Time to start
               #cTargetUnitState := 5;
           ELSE                                                // Stop by no request
               #cTargetUnitState := 0;
           END_IF;
       2:                                                  // PreComfort mode 
           IF #xBlockRequest THEN                               // Stop by alarm      
               #cTargetUnitState := 9;
           ELSIF #xStartRequest THEN                           //Time to start
               #cTargetUnitState := 6;
           ELSE                                                // Stop by no request
               #cTargetUnitState := 0;
           END_IF;
       3:                                                      // Comfort mode 
           IF #xBlockRequest THEN                               // Stop by alarm      
               #cTargetUnitState := 9;
           ELSIF #xStartRequest THEN                           //Time to start
               #cTargetUnitState := 7;
           ELSE                                                // Stop by no request
               #cTargetUnitState := 0;
           END_IF;
       ELSE:
           IF #xBlockRequest THEN                               // Stop by alarm      
               #cTargetUnitState := 9;
           ELSE
               #cTargetUnitState := 0;
           END_IF;
   END_CASE;
END_REGION

REGION Network 2 (SCL)
   IF #cTargetUnitState <> "cTargetUnitStatePrevOne" THEN
       "iTargetUnitStareCounter" := "iTargetUnitStareCounter" + 1;
   END_IF;

   "cTargetUnitStatePrevOne" := #cTargetUnitState;
END_REGION
END_FUNCTION

FUNCTION "AHUActualUnitStatesCtrl" : Void   // FC60105, LAD
{ S7_Optimized_Access := 'TRUE' }
VERSION : 0.1
// Operation Modes                                                 Unit State
// 0=Protection                                                         0=Stopped
// 1=Economy                                                           1=Checking-up  
// 2=PreComfort                                                       2=Preheating
// 3=Comfor                                                              3=Starting 
// 4=Auto(Scheduler)                                              4=RecirculatingOperation
//                                                                                 5=Economy Operation                                                                                                                                            6=PreComfort Operation 
//                                                                                 7=Comfort  operation
//                                                                                 8=Stopping
//                                                                                 9 =Blocking
// stored: AutoNumber false, IsIECCheckEnabled false, SetENOAutomatically false, UDAEnableTagReadback false
   VAR_INPUT
      iUnitID : Int;
      xManualSt1orSt2 : Bool;
      cTargetUnitState : Byte;
      cCheckingUpTime : Byte;
      cPreheatingTime : Byte;
      cStartingTime : Byte;
      cStoppingTime : Byte;
      cWorkOnFullRecycleTime : Byte;
   END_VAR
   VAR_OUTPUT
      cUnitStateForHMI : Byte;
   END_VAR
   VAR_IN_OUT
      cNextUnitState : Byte;
      xActualUnitStateEdge : Bool;
      cCounterToSwitchBtwStates : Int;
   END_VAR
   VAR_TEMP
      cState : Byte;
   END_VAR
BEGIN

REGION Network 1 (SCL)
   CASE #cTargetUnitState OF
       0:
           CASE #cNextUnitState OF
               0:  // 
                   IF #xActualUnitStateEdge THEN
                       #xActualUnitStateEdge := 0;
                   END_IF;
               1..7:  // 
                   #cNextUnitState := 8;
                   #xActualUnitStateEdge := 1;
                   ;
               8:
                   IF #xActualUnitStateEdge THEN
                       #xActualUnitStateEdge := 0;
                       IF #xManualSt1orSt2 THEN
                           #cCounterToSwitchBtwStates := 0;
                       ELSE
                           #cCounterToSwitchBtwStates := #cStoppingTime;
                       END_IF;
                   ELSIF #cCounterToSwitchBtwStates > 0 THEN
                       IF "Timer".x1SecRisingEdge THEN
                           #cCounterToSwitchBtwStates := #cCounterToSwitchBtwStates - 1;
                       END_IF;
                   ELSE
                       #cNextUnitState := 0;
                       #xActualUnitStateEdge := 1;
                   END_IF;
               9:
                   #cNextUnitState := 9;
           END_CASE;
       1..4:
           ;
       5..7:
           CASE #cNextUnitState OF
               0:  // 
                   #cNextUnitState := 1;
                   #xActualUnitStateEdge := 1;
               1:  // 
                   IF #xActualUnitStateEdge THEN
                       #xActualUnitStateEdge := 0;
                       IF #xManualSt1orSt2 THEN
                           #cCounterToSwitchBtwStates := 0;
                       ELSE
                           #cCounterToSwitchBtwStates := #cCheckingUpTime;
                       END_IF;

                   ELSIF #cCounterToSwitchBtwStates > 0 THEN
                       IF "Timer".x1SecRisingEdge THEN
                           #cCounterToSwitchBtwStates := #cCounterToSwitchBtwStates - 1;
                       END_IF;
                   ELSE
                       #cNextUnitState := 2;
                       #xActualUnitStateEdge := 1;
                   END_IF;
               2:
                   IF #xActualUnitStateEdge THEN
                       #xActualUnitStateEdge := 0;
                       IF #xManualSt1orSt2 OR "OAT".Temp.rOAT_Actual > "AHUFrostProt".FrostProt.OATtoStartPreheating[#iUnitID] THEN
                           // Statement section IF
                           #cCounterToSwitchBtwStates := 0;
                       ELSE
                           #cCounterToSwitchBtwStates := #cPreheatingTime;
                       END_IF;
                   ELSIF #cCounterToSwitchBtwStates > 0 THEN
                       IF "Timer".x1SecRisingEdge THEN
                           #cCounterToSwitchBtwStates := #cCounterToSwitchBtwStates - 1;
                       END_IF;
                   ELSE
                       #cNextUnitState := 3;
                       #xActualUnitStateEdge := 1;
                   END_IF;
               3:
                   IF #xActualUnitStateEdge THEN
                       #xActualUnitStateEdge := 0;
                       IF #xManualSt1orSt2 THEN
                           #cCounterToSwitchBtwStates := 0;
                       ELSE
                           #cCounterToSwitchBtwStates := #cStartingTime;
                       END_IF;

                   ELSIF #cCounterToSwitchBtwStates > 0 THEN
                       IF "Timer".x1SecRisingEdge THEN
                           #cCounterToSwitchBtwStates := #cCounterToSwitchBtwStates - 1;
                       END_IF;
                   ELSE
                       #cNextUnitState := 4;
                       #xActualUnitStateEdge := 1;
                   END_IF;
               4:
                   IF #xActualUnitStateEdge THEN
                       #xActualUnitStateEdge := 0;
                       #cCounterToSwitchBtwStates := #cWorkOnFullRecycleTime;
                   ELSIF #cCounterToSwitchBtwStates > 0 THEN
                       IF "Timer".x1SecRisingEdge THEN
                           #cCounterToSwitchBtwStates := #cCounterToSwitchBtwStates - 1;
                       END_IF;
                   ELSE
                       #cNextUnitState := #cTargetUnitState;  // transfer to Econom, PreComf, Comf
                       #xActualUnitStateEdge := 1;
                   END_IF;
               5..7:
                   IF #xActualUnitStateEdge THEN
                       #xActualUnitStateEdge := 0;
                   END_IF;
                   #cNextUnitState := #cTargetUnitState;
               8:
                   #cNextUnitState := 0;
               9:
                   #cNextUnitState := 9;
           END_CASE;
       8:
           ;
       9:
           #cNextUnitState := 9;
   END_CASE;
END_REGION

REGION Network 2 (SCL)
   IF "AHUEqp".Eqp.Cfg.cFan[#iUnitID] > 0 THEN
       IF #cNextUnitState > 2 AND #cNextUnitState < 9 THEN
           #cUnitStateForHMI := 2;
       ELSE
           #cUnitStateForHMI := 1;
       END_IF;
   ELSE
       #cUnitStateForHMI := 0;
   END_IF;
END_REGION
END_FUNCTION

FUNCTION "AHU_Regulation" : Void   // FC60200, FBD
{ S7_Optimized_Access := 'TRUE' }
VERSION : 0.1
// stored: AutoNumber false, IsIECCheckEnabled false, SetENOAutomatically false, UDAEnableTagReadback false
   VAR_INPUT
      iUnitID : Int;   // 1=AHUFood, 2=AHUNonFood
   END_VAR
   VAR_TEMP
      FA_temp : Real;
   END_VAR
BEGIN

REGION Network 1 (SCL): Actual Room (salles area temp)
   // 0=PLC_IO, 1=LoraAvg, 2=MSensor,3 =Auto
   CASE "AHUAI".AI.cRoomTempSelect[#iUnitID] OF
       0:  // 
           "AHUAI".AI.rRoomAirTemp_Actual[#iUnitID] := "AHUAI".AI.rRoomAirTemp_PLC_AI[#iUnitID];
       1:  // 
           "AHUAI".AI.rRoomAirTemp_Actual[#iUnitID] := "AHUAI".AI.rRoomAirTemp_LoraAvg[#iUnitID];
       2: // 
           "AHUAI".AI.rRoomAirTemp_Actual[#iUnitID] := "AHUAI".AI.rRoomAirTemp_MSensor[#iUnitID];
       ELSE
           "AHUAI".AI.rRoomAirTemp_Actual[#iUnitID] := "AHUAI".AI.rRoomAirTemp_PLC_AI[#iUnitID];
   END_CASE;
END_REGION

REGION Network 2: AHUs SetPoints define
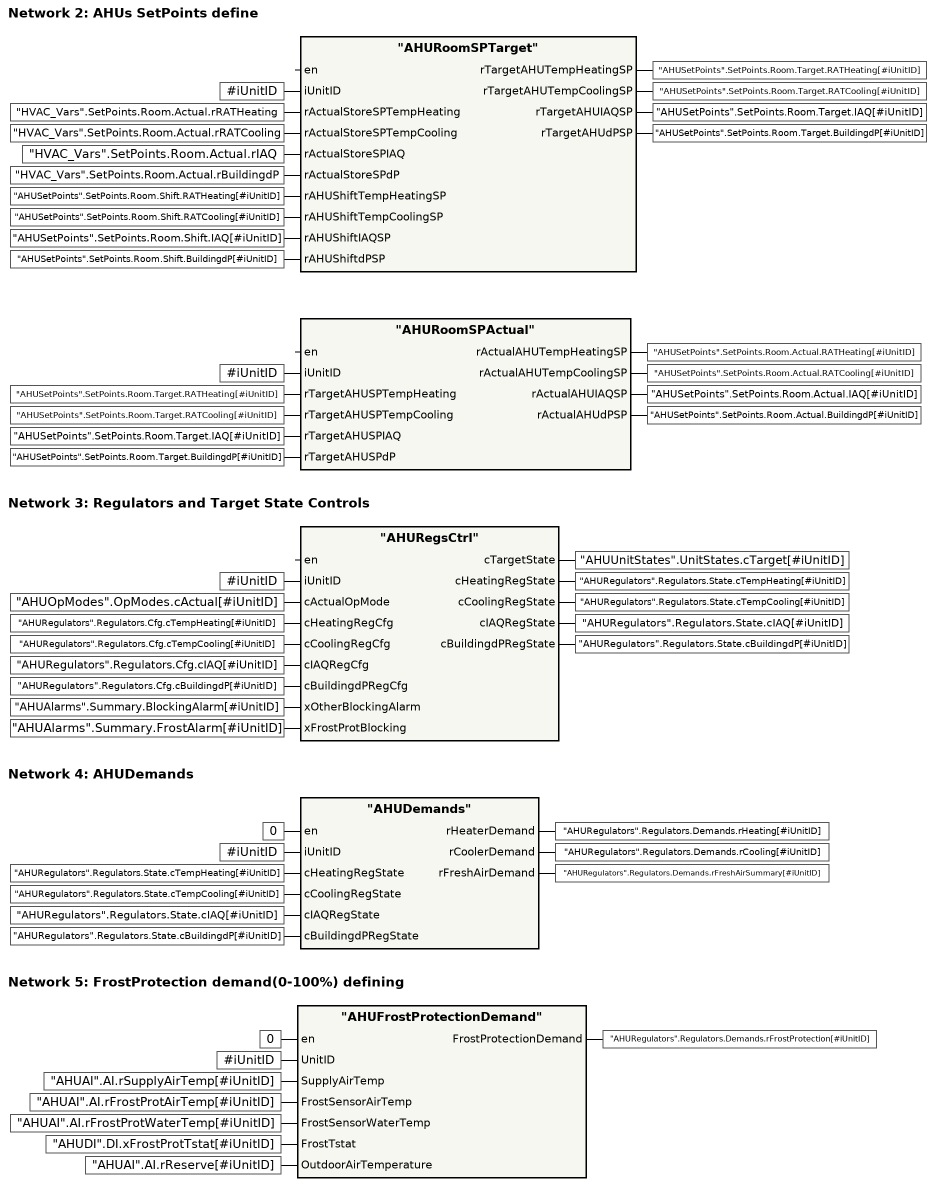
   "AHURoomSPTarget"(iUnitID := #iUnitID,
                     rActualStoreSPTempHeating := "HVAC_Vars".SetPoints.Room.Actual.rRATHeating,
                     rActualStoreSPTempCooling := "HVAC_Vars".SetPoints.Room.Actual.rRATCooling,
                     rActualStoreSPIAQ := "HVAC_Vars".SetPoints.Room.Actual.rIAQ,
                     rActualStoreSPdP := "HVAC_Vars".SetPoints.Room.Actual.rBuildingdP,
                     rAHUShiftTempHeatingSP := "AHUSetPoints".SetPoints.Room.Shift.RATHeating[#iUnitID],
                     rAHUShiftTempCoolingSP := "AHUSetPoints".SetPoints.Room.Shift.RATCooling[#iUnitID],
                     rAHUShiftIAQSP := "AHUSetPoints".SetPoints.Room.Shift.IAQ[#iUnitID],
                     rAHUShiftdPSP := "AHUSetPoints".SetPoints.Room.Shift.BuildingdP[#iUnitID],
                     rTargetAHUTempHeatingSP => "AHUSetPoints".SetPoints.Room.Target.RATHeating[#iUnitID],
                     rTargetAHUTempCoolingSP => "AHUSetPoints".SetPoints.Room.Target.RATCooling[#iUnitID],
                     rTargetAHUIAQSP => "AHUSetPoints".SetPoints.Room.Target.IAQ[#iUnitID],
                     rTargetAHUdPSP => "AHUSetPoints".SetPoints.Room.Target.BuildingdP[#iUnitID]);
   "AHURoomSPActual"(iUnitID := #iUnitID,
                     rTargetAHUSPTempHeating := "AHUSetPoints".SetPoints.Room.Target.RATHeating[#iUnitID],
                     rTargetAHUSPTempCooling := "AHUSetPoints".SetPoints.Room.Target.RATCooling[#iUnitID],
                     rTargetAHUSPIAQ := "AHUSetPoints".SetPoints.Room.Target.IAQ[#iUnitID],
                     rTargetAHUSPdP := "AHUSetPoints".SetPoints.Room.Target.BuildingdP[#iUnitID],
                     rActualAHUTempHeatingSP => "AHUSetPoints".SetPoints.Room.Actual.RATHeating[#iUnitID],
                     rActualAHUTempCoolingSP => "AHUSetPoints".SetPoints.Room.Actual.RATCooling[#iUnitID],
                     rActualAHUIAQSP => "AHUSetPoints".SetPoints.Room.Actual.IAQ[#iUnitID],
                     rActualAHUdPSP => "AHUSetPoints".SetPoints.Room.Actual.BuildingdP[#iUnitID]);
END_REGION

REGION Network 3: Regulators and Target State Controls
   "AHURegsCtrl"(iUnitID := #iUnitID,
                 cActualOpMode := "AHUOpModes".OpModes.cActual[#iUnitID],
                 cHeatingRegCfg := "AHURegulators".Regulators.Cfg.cTempHeating[#iUnitID],
                 cCoolingRegCfg := "AHURegulators".Regulators.Cfg.cTempCooling[#iUnitID],
                 cIAQRegCfg := "AHURegulators".Regulators.Cfg.cIAQ[#iUnitID],
                 cBuildingdPRegCfg := "AHURegulators".Regulators.Cfg.cBuildingdP[#iUnitID],
                 xOtherBlockingAlarm := "AHUAlarms".Summary.BlockingAlarm[#iUnitID],
                 xFrostProtBlocking := "AHUAlarms".Summary.FrostAlarm[#iUnitID],
                 cTargetState => "AHUUnitStates".UnitStates.cTarget[#iUnitID],
                 cHeatingRegState => "AHURegulators".Regulators.State.cTempHeating[#iUnitID],
                 cCoolingRegState => "AHURegulators".Regulators.State.cTempCooling[#iUnitID],
                 cIAQRegState => "AHURegulators".Regulators.State.cIAQ[#iUnitID],
                 cBuildingdPRegState => "AHURegulators".Regulators.State.cBuildingdP[#iUnitID]);
END_REGION

REGION Network 4: AHUDemands
   // Regulator State -> Demands
   IF 0 THEN
       "AHUDemands"(iUnitID := #iUnitID,
                    cHeatingRegState := "AHURegulators".Regulators.State.cTempHeating[#iUnitID],
                    cCoolingRegState := "AHURegulators".Regulators.State.cTempCooling[#iUnitID],
                    cIAQRegState := "AHURegulators".Regulators.State.cIAQ[#iUnitID],
                    cBuildingdPRegState := "AHURegulators".Regulators.State.cBuildingdP[#iUnitID],
                    rHeaterDemand => "AHURegulators".Regulators.Demands.rHeating[#iUnitID],
                    rCoolerDemand => "AHURegulators".Regulators.Demands.rCooling[#iUnitID],
                    rFreshAirDemand => "AHURegulators".Regulators.Demands.rFreshAirSummary[#iUnitID]);
   END_IF;
END_REGION

REGION Network 5: FrostProtection demand(0-100%) defining
   IF 0 THEN
       "AHUFrostProtectionDemand"(UnitID := #iUnitID,
                               SupplyAirTemp := "AHUAI".AI.rSupplyAirTemp[#iUnitID],
                               FrostSensorAirTemp := "AHUAI".AI.rFrostProtAirTemp[#iUnitID],
                               FrostSensorWaterTemp := "AHUAI".AI.rFrostProtWaterTemp[#iUnitID],
                               FrostTstat := "AHUDI".DI.xFrostProtTstat[#iUnitID],
                               OutdoorAirTemperature := "AHUAI".AI.rReserve[#iUnitID],
                               FrostProtectionDemand => "AHURegulators".Regulators.Demands.rFrostProtection[#iUnitID]);
   END_IF;
END_REGION
END_FUNCTION

FUNCTION "AHURoomSPTarget" : Void   // FC60006, LAD
{ S7_Optimized_Access := 'TRUE' }
VERSION : 0.1
// stored: AutoNumber false, IsIECCheckEnabled false, SetENOAutomatically false, UDAEnableTagReadback false
   VAR_INPUT
      iUnitID : Int;
      rActualStoreSPTempHeating : Real;
      rActualStoreSPTempCooling : Real;
      rActualStoreSPIAQ : Real;
      rActualStoreSPdP : Real;
      rAHUShiftTempHeatingSP : Real;
      rAHUShiftTempCoolingSP : Real;
      rAHUShiftIAQSP : Real;
      rAHUShiftdPSP : Real;
   END_VAR
   VAR_OUTPUT
      rTargetAHUTempHeatingSP : Real;
      rTargetAHUTempCoolingSP : Real;
      rTargetAHUIAQSP : Real;
      rTargetAHUdPSP : Real;
   END_VAR
   VAR_TEMP
      iTargetUnitMode_old : Int;
      xResetActualOperationMode : Bool;
      iActualUnitMode_old : Int;
      xResetTargetSetpoints : Bool;
   END_VAR
BEGIN

REGION Network 1 (SCL)
   #rTargetAHUTempHeatingSP := #rActualStoreSPTempHeating + #rAHUShiftTempHeatingSP;
   #rTargetAHUTempCoolingSP := #rActualStoreSPTempCooling + #rAHUShiftTempCoolingSP;
   #rTargetAHUIAQSP := #rActualStoreSPIAQ + #rAHUShiftIAQSP;
   #rTargetAHUdPSP := #rActualStoreSPdP + #rAHUShiftdPSP;
END_REGION
END_FUNCTION

FUNCTION "AHURoomSPActual" : Void   // FC60005, LAD
{ S7_Optimized_Access := 'TRUE' }
VERSION : 0.1
// stored: AutoNumber false, IsIECCheckEnabled false, SetENOAutomatically false, UDAEnableTagReadback false
   VAR_INPUT
      iUnitID : Int;
      rTargetAHUSPTempHeating : Real;
      rTargetAHUSPTempCooling : Real;
      rTargetAHUSPIAQ : Real;
      rTargetAHUSPdP : Real;
   END_VAR
   VAR_OUTPUT
      rActualAHUTempHeatingSP : Real;
      rActualAHUTempCoolingSP : Real;
      rActualAHUIAQSP : Real;
      rActualAHUdPSP : Real;
   END_VAR
   VAR_TEMP
      iTargetUnitMode_old : Int;
      xResetActualOperationMode : Bool;
      iActualUnitMode_old : Int;
      xResetTargetSetpoints : Bool;
   END_VAR
BEGIN

REGION Network 1 (SCL): Smoothing Actual Setpoints
   IF 1 THEN
       #rActualAHUTempHeatingSP := "AHUSetPoints".SetPoints.Room.Target.RATHeating[#iUnitID];
       #rActualAHUTempCoolingSP := "AHUSetPoints".SetPoints.Room.Target.RATCooling[#iUnitID];
       #rActualAHUIAQSP := "AHUSetPoints".SetPoints.Room.Target.IAQ[#iUnitID];
       #rActualAHUdPSP := "AHUSetPoints".SetPoints.Room.Target.BuildingdP[#iUnitID];
   END_IF;
END_REGION
END_FUNCTION

FUNCTION "AHURegsCtrl" : Void   // FC60030, LAD
{ S7_Optimized_Access := 'TRUE' }
VERSION : 0.1
// Operation Modes                                                 Unit State
// 0=Protection                                                         0=Stopped
// 1=Economy                                                           1=Checking-up  
// 2=PreComfort                                                       2=Preheating
// 3=Comfor                                                              3=Starting 
// 4=Auto(Scheduler)                                              4=RecirculatingOperation (Protection)
//                                                                                 5=Sustained Mode (Economy setpoints)
//                                                                                 6=Sustained Mode (PreComfort setpoints) 
//                                                                                 7=Comfort  operation
//                                                                                 8=Stopping
//                                                                                 9=Blocking
// stored: AutoNumber false, IsIECCheckEnabled false, SetENOAutomatically false, UDAEnableTagReadback false
   VAR_INPUT
      iUnitID : Int;
      cActualOpMode : Byte;
      cHeatingRegCfg : Byte;
      cCoolingRegCfg : Byte;
      cIAQRegCfg : Byte;
      cBuildingdPRegCfg : Byte;
      xOtherBlockingAlarm : Bool;
      xFrostProtBlocking : Bool;
   END_VAR
   VAR_OUTPUT
      cTargetState : Byte;
      cHeatingRegState : Byte;
      cCoolingRegState : Byte;
      cIAQRegState : Byte;
      cBuildingdPRegState : Byte;
   END_VAR
   VAR_TEMP
      cActualOpModeSequence : Byte;   // Поточний цикл
   END_VAR
BEGIN

REGION Network 1 (SCL)
   IF #xFrostProtBlocking THEN
       // Frost protection
       #cTargetState := 11;
   ELSIF #xOtherBlockingAlarm THEN
       // Blocking Alarm
       #cTargetState := 10;
   ELSE
       CASE #cActualOpMode OF
           0:  // Protection 
               "AHURegsAndTargetStatesInProtectionOpMode"(iUnitID:=#iUnitID,
                                                          cActualOpMode:=#cActualOpMode,
                                                          cHeatingRegCfg:=#cHeatingRegCfg,
                                                          cCoolingRegCfg:=#cCoolingRegCfg,
                                                          cIAQRegCfg:=#cIAQRegCfg,
                                                          cBuildingdPRegCfg:=#cBuildingdPRegCfg,
                                                          cTargetState=>#cTargetState,
                                                          cHeatingRegState=>#cHeatingRegState,
                                                          cCoolingRegState=>#cCoolingRegState,
                                                          cIAQRegState=>#cIAQRegState,
                                                          cBuildingdPRegState=>#cBuildingdPRegState);

           1:  // Economy
               "AHURegsAndTargetStatesInEconomyOpMode"(iUnitID:=#iUnitID,
                                                       cActualOpMode:=#cActualOpMode,
                                                       cHeatingRegCfg:=#cHeatingRegCfg,
                                                       cCoolingRegCfg:=#cCoolingRegCfg,
                                                       cIAQRegCfg:=#cIAQRegCfg,
                                                       cBuildingdPRegCfg:=#cBuildingdPRegCfg,
                                                       cTargetState=>#cTargetState,
                                                       cHeatingRegState=>#cHeatingRegState,
                                                       cCoolingRegState=>#cCoolingRegState,
                                                       cIAQRegState=>#cIAQRegState,
                                                       cBuildingdPRegState=>#cBuildingdPRegState);
           2: // PreComfort
               "AHURegsAndTargetStatesInPreComfortOpMode"(iUnitID:=#iUnitID,
                                                          cActualOpMode:=#cActualOpMode,
                                                          cHeatingRegCfg:=#cHeatingRegCfg,
                                                          cCoolingRegCfg:=#cCoolingRegCfg,
                                                          cIAQRegCfg:=#cIAQRegCfg,
                                                          cBuildingdPRegCfg:=#cBuildingdPRegCfg,
                                                          cTargetState=>#cTargetState,
                                                          cHeatingRegState=>#cHeatingRegState,
                                                          cCoolingRegState=>#cCoolingRegState,
                                                          cIAQRegState=>#cIAQRegState,
                                                          cBuildingdPRegState=>#cBuildingdPRegState);
           ELSE  //Comfort
               "AHURegsAndTargetStatesInComfortOpMode"(iUnitID:=#iUnitID,
                                                       cActualOpMode:=#cActualOpMode,
                                                       cHeatingRegCfg:=#cHeatingRegCfg,
                                                       cCoolingRegCfg:=#cCoolingRegCfg,
                                                       cIAQRegCfg:=#cIAQRegCfg,
                                                       cBuildingdPRegCfg:=#cBuildingdPRegCfg,
                                                       cTargetState=>#cTargetState,
                                                       cHeatingRegState=>#cHeatingRegState,
                                                       cCoolingRegState=>#cCoolingRegState,
                                                       cIAQRegState=>#cIAQRegState,
                                                       cBuildingdPRegState=>#cBuildingdPRegState);
       END_CASE;
       ;
   END_IF;
END_REGION
END_FUNCTION

FUNCTION "AHUDemands" : Void   // FC60008, LAD
{ S7_Optimized_Access := 'TRUE' }
VERSION : 0.1
// stored: AutoNumber false, IsIECCheckEnabled false, SetENOAutomatically false, UDAEnableTagReadback false
   VAR_INPUT
      iUnitID : Int;
      cHeatingRegState : Byte;
      cCoolingRegState : Byte;
      cIAQRegState : Byte;
      cBuildingdPRegState : Byte;
   END_VAR
   VAR_OUTPUT
      rHeaterDemand : Real;
      rCoolerDemand : Real;
      rFreshAirDemand : Real;
   END_VAR
BEGIN

REGION Network 1: Temperature demands(0-100%) defining (PID)
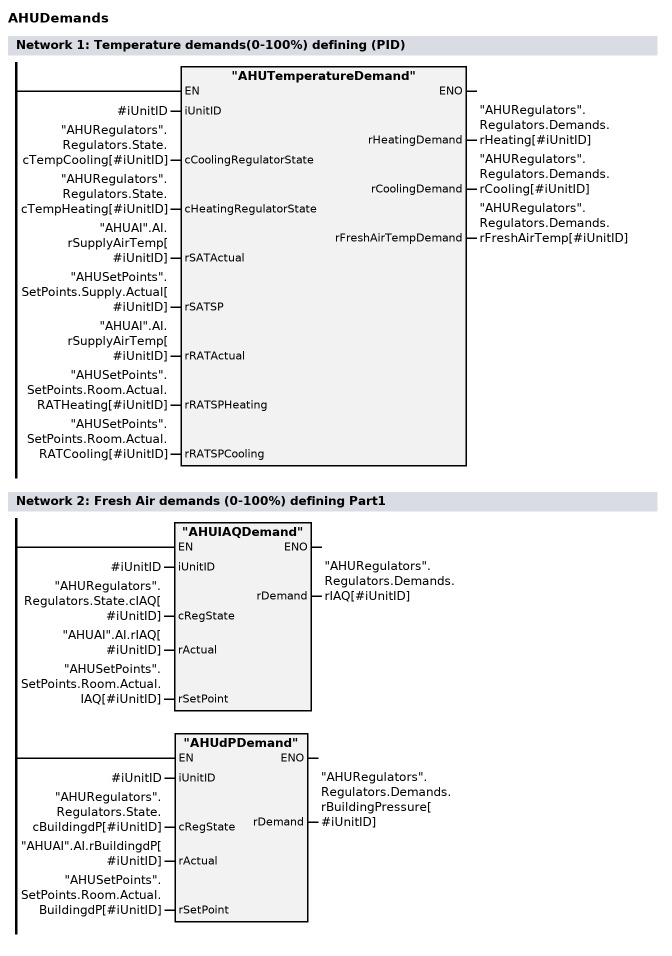
   RUNG wire#powerrail
      "AHUTemperatureDemand"(iUnitID := #iUnitID, cCoolingRegulatorState := "AHURegulators".Regulators.State.cTempCooling[#iUnitID], cHeatingRegulatorState := "AHURegulators".Regulators.State.cTempHeating[#iUnitID], rSATActual := "AHUAI".AI.rSupplyAirTemp[#iUnitID], rSATSP := "AHUSetPoints".SetPoints.Supply.Actual[#iUnitID], rRATActual := "AHUAI".AI.rSupplyAirTemp[#iUnitID], rRATSPHeating := "AHUSetPoints".SetPoints.Room.Actual.RATHeating[#iUnitID], rRATSPCooling := "AHUSetPoints".SetPoints.Room.Actual.RATCooling[#iUnitID], rHeatingDemand => "AHURegulators".Regulators.Demands.rHeating[#iUnitID], rCoolingDemand => "AHURegulators".Regulators.Demands.rCooling[#iUnitID], rFreshAirTempDemand => "AHURegulators".Regulators.Demands.rFreshAirTemp[#iUnitID])
   END_RUNG
   // the same network as SCL:
   "AHUTemperatureDemand"(iUnitID := #iUnitID,
                          cCoolingRegulatorState := "AHURegulators".Regulators.State.cTempCooling[#iUnitID],
                          cHeatingRegulatorState := "AHURegulators".Regulators.State.cTempHeating[#iUnitID],
                          rSATActual := "AHUAI".AI.rSupplyAirTemp[#iUnitID],
                          rSATSP := "AHUSetPoints".SetPoints.Supply.Actual[#iUnitID],
                          rRATActual := "AHUAI".AI.rSupplyAirTemp[#iUnitID],
                          rRATSPHeating := "AHUSetPoints".SetPoints.Room.Actual.RATHeating[#iUnitID],
                          rRATSPCooling := "AHUSetPoints".SetPoints.Room.Actual.RATCooling[#iUnitID],
                          rHeatingDemand => "AHURegulators".Regulators.Demands.rHeating[#iUnitID],
                          rCoolingDemand => "AHURegulators".Regulators.Demands.rCooling[#iUnitID],
                          rFreshAirTempDemand => "AHURegulators".Regulators.Demands.rFreshAirTemp[#iUnitID]);
END_REGION

REGION Network 2: Fresh Air demands (0-100%) defining Part1
   RUNG wire#powerrail
      "AHUIAQDemand"(iUnitID := #iUnitID, cRegState := "AHURegulators".Regulators.State.cIAQ[#iUnitID], rActual := "AHUAI".AI.rIAQ[#iUnitID], rSetPoint := "AHUSetPoints".SetPoints.Room.Actual.IAQ[#iUnitID], rDemand => "AHURegulators".Regulators.Demands.rIAQ[#iUnitID])
   END_RUNG
   RUNG wire#powerrail
      "AHUdPDemand"(iUnitID := #iUnitID, cRegState := "AHURegulators".Regulators.State.cBuildingdP[#iUnitID], rActual := "AHUAI".AI.rBuildingdP[#iUnitID], rSetPoint := "AHUSetPoints".SetPoints.Room.Actual.BuildingdP[#iUnitID], rDemand => "AHURegulators".Regulators.Demands.rBuildingPressure[#iUnitID])
   END_RUNG
   // the same network as SCL:
   "AHUIAQDemand"(iUnitID := #iUnitID,
                  cRegState := "AHURegulators".Regulators.State.cIAQ[#iUnitID],
                  rActual := "AHUAI".AI.rIAQ[#iUnitID],
                  rSetPoint := "AHUSetPoints".SetPoints.Room.Actual.IAQ[#iUnitID],
                  rDemand => "AHURegulators".Regulators.Demands.rIAQ[#iUnitID]);
   "AHUdPDemand"(iUnitID := #iUnitID,
                 cRegState := "AHURegulators".Regulators.State.cBuildingdP[#iUnitID],
                 rActual := "AHUAI".AI.rBuildingdP[#iUnitID],
                 rSetPoint := "AHUSetPoints".SetPoints.Room.Actual.BuildingdP[#iUnitID],
                 rDemand => "AHURegulators".Regulators.Demands.rBuildingPressure[#iUnitID]);
END_REGION

REGION Network 3 (SCL): Fresh Air demands defining Part2
   (* "AHUDmnds".Demands.rFreshAir[#iUnitID] := MAX(IN1 := "AHUDmnds".Demands.rIAQ[#iUnitID] * "AHUFreshAirCoef".FreshAirCoef.IAQ[#iUnitID],
                                                IN2 := "AHUDmnds".Demands.rBuildingPressure[#iUnitID] * "AHUFreshAirCoef".FreshAirCoef.BuildingdP[#iUnitID],
                                                IN3 := "AHUDmnds".Demands.rFreshAirTemp[#iUnitID] * "AHUFreshAirCoef".FreshAirCoef.Temperature[#iUnitID]); *)
END_REGION
END_FUNCTION

